IF (OP80_HMI_AutoMode AND NOT OP80_HMI_ManualMOde AND NOT OP80_HMI_StepMode) THEN
		OP80_Modeselection_FB.ModeWord:=1;
	ELSIF (NOT OP80_HMI_AutoMode AND OP80_HMI_ManualMOde AND NOT OP80_HMI_StepMode) THEN
		OP80_Modeselection_FB.ModeWord:=2;
	ELSIF  (NOT OP80_HMI_AutoMode AND NOT OP80_HMI_ManualMOde AND  OP80_HMI_StepMode) THEN
		OP80_Modeselection_FB.ModeWord:=3;
    ELSE   
		OP80_Modeselection_FB.ModeWord:=0;
END_IF
OP80_Modeselection_FB(
	ModeWord:= , 
	HomeConditionOK:=OP80_HomeConditionOK , 
	OperationEnable:=OP80_AutoSelected, 
	StartPB:=OP80_HMI_CycleStart , 
	SafetyAndNOError:= OP80_Safety_OK, 
	ModeAck:=TRUE , 
	HomingINProgress:=OP80_HomeRunning , 
	TempHomeOK:=OP80_Temp_hmeOK , 
	ResetPB:= , 
	AutoSelected=> OP80_AutoSelected, 
	ManualSelected=> OP80_ManualSelected, 
	StepSelected=>OP80_StepSelected , 
	ModeSelAck_Indication=> , 
	StatusDisplay=> , 
	AutoRunning:=OP80_AutoRunning, 
	StepRunning:=OP80_StepRunning , 
	StartEnable:=OP80_StartEnable  , 
	MachineStop:=OP80_Machine_Stop );

OP80_Safety_OK:=OperationEnable;	
	
IF OP80_AutoSelected OR OP80_ManualSelected AND NOT ( OP80_ErrorActive OR OP80_Safety_OK) THEN
	SR60_Vert_servo.bEnable:=TRUE;
ELSE
	SR60_Vert_servo.bEnable:=FALSE;
END_IF

IF SR80_Vert_servo.bAxisError OR NOT OP80_Safety_OK  THEN
	OP80_ErrorActive:=TRUE;
END_IF

OP80_Safety_OK:=OperationEnable;

IF OP80_Stop_Request AND NOT OP80_STN_ENABLE THEN
	OP80_Machine_Stop:=1;
END_IF
Gen_Timer(IN:=OP80_Machine_Stop,PT:=T#5S);
IF Gen_Timer.Q THEN
	OP80_Machine_Stop:=0;
END_IF

END_PROGRAM

// ---- POUs/Programs/OP80/OP80_MANUAL.TcPOU
PROGRAM OP80_MANUAL
VAR
	//SR80_Vert_servo_status:stManualModeAxis;
	SR80_Vert_servo_Axis :AXIS_REF;
    temp_safe:BOOL;
	enable:BOOL;
	reset:bool;
	Op80Enable: BOOL;
END_VAR


// IF MANUAL IS SELECTED 

//SR80_Vert_servo_ctrl.ABSmove_Start:=OP80_VERT_SERVO_STRT;
//OP80_SERVO_POS_DONE:= SR80_Vert_servo_ctrl.pos_done;

IF In_Range(SR80_Vert_servo_status.actualPosition,OP80_VERT_SERVO_SFE_WRK_POS,1) THEN
	OP80_SERVO_ON_SFE_WRK := TRUE;
ELSE
	OP80_SERVO_ON_SFE_WRK := FALSE;
END_IF

IF In_Range(SR80_Vert_servo_status.actualPosition,OP80_VERT_SERVO_HME_POS,1) THEN
	OP80_SERVO_ON_HOME := TRUE;
ELSE
	OP80_SERVO_ON_HOME := FALSE;
END_IF

IF In_Range(SR80_Vert_servo_status.actualPosition,OP80_VERT_SERVO_WRK_POS_1,1) THEN
	OP80_SERVO_ON_WRK_1 := TRUE;
ELSE
	OP80_SERVO_ON_WRK_1 := FALSE;
END_IF

IF In_Range(SR80_Vert_servo_status.actualPosition,OP80_VERT_SERVO_WRK_POS_2,1) THEN
	OP80_SERVO_ON_WRK_2 := TRUE;
ELSE
	OP80_SERVO_ON_WRK_2 := FALSE;
END_IF

OP80_VERT_SERVO_SFE_WRK_POS   :=  OP80_HMI_Safe_Work;
OP80_VERT_SERVO_HME_POS       :=  OP80_HMI_Safe_Home;
OP80_VERT_SERVO_WRK_POS_2     :=  OP80_VERT_SERVO_WORK_POS;
OP80_VERT_SERVO_WRK_POS_1	  := (OP80_VERT_SERVO_WRK_POS_2-OP80_HMI_Servo_Pos_Offset);

SR80_Vert_servo(
	bAxis1_Ref_Switch:= , 
	bInit:= , 
	bErrorReset:= OP80_HMI_Reset OR Servo_Reset , 
	bEnable:= Servo_Enable, 
	bMoveVelocity:= , 
	bHalt:= , 
	bManualMode:=OP80_ManualSelected AND MANUAL_SELECTED , 
	fHomePos:= , 
	fOverride:= , 
	fTargetPosition:=SR80_Vert_servo_ctrl.Position , 
	fTargetVelocity:=SR80_Vert_servo_ctrl.Velocity , 
	fAcc:= , 
	fDec:= , 
	Servo_High_Limit:= OP80_HMI_High_Limit,	
	Servo_Low_Limit:=  OP80_HMI_Low_Limit,	
	Safe_move_Conditions:=Servo_Safety,
	Axis:=SR80_Vert_servo_Axis  , 
	bmove_home:=SR80_Vert_servo_ctrl.Axis_Home_Cmd ,
	baxis_in_home_pos=>SR80_Vert_servo_ctrl.Axis_In_Home ,
	HME_WRITE_ADD:= 16#500F,	
	bHome:=SR80_Vert_servo_ctrl.Bsethome , 
	bSetPosition:=SR80_Vert_servo_ctrl.BsetPos , 
	bMoveAbsolute:=SR80_Vert_servo_ctrl.ABSmove_Start , 
	bMoveRelative:=SR80_Vert_servo_ctrl.RELmove_Start ,
	bMoveTorque :=SR80_Vert_servo_ctrl.Torque_mode_Start,
	stManualModeAxis:=SR80_Vert_servo_status , 
	sAxisState=>SR80_Vert_servo_ctrl.Axis_State , 
	bAxis_ready=>SR80_Vert_servo_ctrl.Axis_ready , 
	bAxisInPosition=> SR80_Vert_servo_ctrl.Axis_In_Pos, 
	bAxisError=>SR80_Vert_servo_ctrl.Axis_Error , 
	bAxisEnabled=> SR80_Vert_servo_ctrl.Axis_Enabled, 
	bAxisHomed=> SR80_Vert_servo_ctrl.Axis_reference, 
	bSetPositionDone=>   ,
    bsafe_to_move=>SR80_Vert_servo_ctrl.Safe_To_Move,  
	bABS_Pos_done=> SR80_Vert_servo_ctrl.pos_done,
	Actual_position=>SR80_Vert_servo_ctrl.Actual_Position ,  
	Actual_velocity=>SR80_Vert_servo_ctrl.Actual_Velocity , 
	Actual_Torque=> SR80_Vert_servo_ctrl.Actual_Torque,	
	bHaltDone=> , 
	bSTOPDone=> , 
	bHomeDone=> , 
	bDone=> );
	
IF MANUAL_SELECTED AND OP80_ManualSelected THEN
	SR80_Vert_servo_status.targetVelocity:=50;	
END_IF

OP80_LH_LVDT_VALUE := DINT_TO_REAL(OP80_LH)/10000;
OP80_RH_LVDT_VALUE := DINT_TO_REAL(OP80_RH)/10000;

END_PROGRAM

// ---- POUs/Programs/OP80/OP80_AUTOSEQUENCE.TcPOU
PROGRAM OP80_AUTOSEQUENCE
VAR

//INT

	OP80_FIXTURE_2					: INT;
	OP80_FIXTURE_1					: INT;	
	Dry_run : BOOL;
// TIMER
	OP80_AFT_WRK_POS : TON;
	
	check: BOOL;
	OP80_STN_MOVER: INT;
	OP80_Cycle_Time_FB : FB_Cycletime;
	MOVER_POS_RECHED_R: R_TRIG;
END_VAR

VAR PERSISTENT

END_VAR

IF (NOT OP80_AutoSelected) OR (OP80_ErrorActive OR OP80_HomeRunning ) OR NOT OperationEnable THEN
	OP80_AutoRunning:= FALSE;
	OP80_AutoSeq:= 10;
END_IF	


CASE OP80_AutoSeq OF
		
		10: IF (OP80_AutoSelected) THEN		// Check Automode Selected
				OP80_AutoSeq:=20;
	        END_IF
		
	    20:IF ( NOT OP80_ErrorActive) THEN		//Check No error
		       OP80_AutoSeq:=30;
      	   END_IF
		   
      	30:IF (NOT OP80_HomeRunning) THEN		//Check No Homerunning
      		   OP80_AutoSeq :=40;
      	   END_IF
		   
        40:IF (OP80_Main.OP80_Modeselection_FB.TempHomeOK)THEN	//Check Machine in Home
      		   OP80_AutoSeq:= 50;
      	   END_IF
		   
      	50:IF ( OP80_STN_ENABLE AND OP80_STN_RUNNING ) THEN		// Check Operation Completed Reset
      		   OP80_AutoSeq:=70;
		   ELSE
	   		   OP80_AutoSeq:=60;
      	   END_IF
		   
	   60:IF (AUTO_RUNNING OR (NOT AUTO_RUNNING AND OP80_HMI_CycleStart)) THEN		//Machine Start in Fully Automatic or Press Cycle Start For Semi Automatic
		    OP80_HomeConditionOK:=TRUE;
	 			IF( OP80_Main.OP80_Modeselection_FB.HomeConditionOK AND OP80_AutoSelected) THEN
					OP80_AutoRunning:=TRUE;
					OP80_StepRunning:= FALSE;		
				ELSIF (OP80_Main.OP80_Modeselection_FB.HomeConditionOK AND OP80_StepSelected) THEN
					OP80_AutoRunning:=FALSE;
					OP80_StepRunning:= TRUE;
				END_IF;
		  END_IF
		  
		  IF ((OP80_AutoRunning OR OP80_StepRunning) AND OP80_StartEnable) THEN
			OP80_AutoSeq:= 70;
		  END_IF	

      	70:  // SERVO POSITION SAFE CHECK
	       IF (OP80_SERVO_ON_SFE_WRK OR OP80_SERVO_ON_HOME) AND NOT SR80_Vert_servo_ctrl.ABSmove_Start THEN 
	        SR80_Vert_servo_ctrl.Position:=OP80_VERT_SERVO_WRK_POS_1;   
	        OP80_AutoSeq:=75;
	       END_IF
		   
		75: // WAITING FOR MOVER AND MOVING SERVO TO TARGET POSITION
			IF OP80_STN_ENABLE AND SR80_Vert_servo_ctrl.Position=OP80_VERT_SERVO_WRK_POS_1 THEN
			 SR80_Vert_servo_ctrl.Velocity:=OP80_HMI_Servo_Speed;
			 OP80_STN_RUNNING:=1;
			 SR80_Vert_servo_ctrl.ABSmove_Start:=TRUE;
			 IF OP80_FIXTURE_1=70 OR OP80_FIXTURE_2=70 THEN
			 	OP80_AutoSeq:=80;
			 ELSIF OP80_FIXTURE_1<>70 AND OP80_FIXTURE_2<>70 THEN
				OP80_AutoSeq:=76;
			 END_IF	
			END_IF

		 76:OP80_STN_ENABLE:=0;
			IF 	(MOVER_CMP_STATUS[OP80_STN_MOVER][1]=71 AND MOVER_CMP_STATUS[OP80_STN_MOVER][2]=71) THEN
				MOVER_STP_NO[OP80_CURR_MOVER]	:= (OP80_XTS_POS_NO*10);
			ELSE		
				STATION_DONE[OP80_CURR_MOVER][OP80_XTS_POS_NO]	:= TRUE;
			END_IF	
			IF MOVER_STP_NO[OP80_CURR_MOVER]<>((OP80_XTS_POS_NO*10)+1)THEN 
				OP80_CURR_MOVER	:= 0;
				OP80_AutoSeq	:= 76;  
			END_IF	
			
		80:  IF SR80_Vert_servo_ctrl.pos_done AND OP80_SERVO_ON_WRK_1 THEN
			   SR80_Vert_servo_ctrl.ABSmove_Start:=FALSE;
			   SR80_Vert_servo_ctrl.Position:=OP80_GVL.OP80_VERT_SERVO_WRK_POS_2;
			   SR80_Vert_servo_ctrl.Velocity:=(OP80_HMI_Servo_Speed-OP80_HMI_Servo_Speed_Offset);
			   OP80_AutoSeq:=90;
			 ELSIF SR80_Vert_servo_ctrl.pos_done AND OP80_SERVO_ON_WRK_2 THEN
 				OP80_AutoSeq:=100;
			 END_IF
			  
		90: IF OP80_SERVO_ON_WRK_1 AND NOT SR80_Vert_servo_ctrl.ABSmove_Start THEN                   
               SR80_Vert_servo_ctrl.ABSmove_Start:=TRUE;
				OP80_LH_LVDT_OK:=0;
				OP80_LH_LVDT_NOK:=0;
				OP80_RH_LVDT_OK:=0;
				OP80_RH_LVDT_NOK:=0; 
               OP80_AutoSeq:=100;
			END_IF
			
		100: // START THE SPINNER OK COMPONENT FIXTURE
			IF OP80_AFT_WRK_POS.Q AND OP80_SERVO_ON_WRK_2 THEN	
			 SR80_Vert_servo_ctrl.ABSmove_Start:=FALSE;		 
			  IF OP80_FIXTURE_1=70 THEN
			 	 IF In_Range(OP80_LH_LVDT_VALUE,OP80_SET_LVDT_VALUE,OP80_LVDT_TOLERANCE) THEN
				  OP80_LH_LVDT_OK  := 1;
				  OP80_LH_LVDT_NOK := 0;				  				  
			 	 ELSE
				  OP80_LH_LVDT_NOK := 1;
				  OP80_LH_LVDT_OK  := 0;
			 	 END_IF  
			  END_IF
			  IF OP80_FIXTURE_2=70 THEN
			  	IF In_Range(OP80_RH_LVDT_VALUE,OP80_SET_LVDT_VALUE,OP80_LVDT_TOLERANCE) THEN
				  OP80_RH_LVDT_OK  := 1;
				  OP80_RH_LVDT_NOK := 0;			  				  
			  	ELSE
				  OP80_RH_LVDT_NOK := 1;
				  OP80_RH_LVDT_OK  := 0;
			    END_IF
		 	  END_IF
				OP80_HMI_LH_LVDT_VALUE:=OP80_LH_LVDT_VALUE;
				OP80_HMI_RH_LVDT_VALUE:=OP80_RH_LVDT_VALUE;				  
			  IF NOT SR80_Vert_servo_ctrl.ABSmove_Start THEN
				 SR80_Vert_servo_ctrl.Position:=OP80_VERT_SERVO_SFE_WRK_POS;
				 SR80_Vert_servo_ctrl.Velocity:=OP80_HMI_Servo_Speed;
				 OP80_STN_ENABLE:=FALSE;
				 OP80_AutoSeq:=110;
			  END_IF				    			  
		    END_IF
			OP80_CURR_MOVER			:= OP80_STN_MOVER;
		
		110: // SERVO MOVE TO SAFE WORK POSITION	 
			IF NOT SR80_Vert_servo_ctrl.ABSmove_Start AND SR80_Vert_servo.fTargetPosition=OP80_VERT_SERVO_SFE_WRK_POS THEN
				SR80_Vert_servo_ctrl.ABSmove_Start:=TRUE;
				IF OP80_LH_LVDT_OK THEN
					MOVER_CMP_STATUS[OP80_CURR_MOVER][1]:=80;
				ELSIF OP80_LH_LVDT_NOK THEN  
					MOVER_CMP_STATUS[OP80_CURR_MOVER][1]:=81;	
				END_IF
				IF OP80_RH_LVDT_OK THEN
					MOVER_CMP_STATUS[OP80_CURR_MOVER][2]:=80;
				ELSIF OP80_RH_LVDT_NOK THEN  
					MOVER_CMP_STATUS[OP80_CURR_MOVER][2]:=81;	
				END_IF									
				OP80_AutoSeq:=120;
			END_IF

				
		120: // SERVO DONE
			IF SR80_Vert_servo_ctrl.pos_done AND OP80_SERVO_ON_SFE_WRK THEN
			 	SR80_Vert_servo_ctrl.ABSmove_Start:=FALSE;
				OP80_STN_ENABLE:=0;				
			 	OP80_AutoSeq:=70;
				OP80_STN_RUNNING:=0;
			IF (MOVER_CMP_STATUS[OP80_CURR_MOVER][1]=81 AND MOVER_CMP_STATUS[OP80_CURR_MOVER][2]=81) THEN	
				MOVER_STP_NO[OP80_CURR_MOVER]	:= (OP160_XTS_POS_NO*10);
			ELSE
			STATION_DONE[OP80_CURR_MOVER][OP80_XTS_POS_NO]			:= TRUE;
		   END_IF	
		END_IF		
END_CASE 

OP80_Cycle_Time_FB(i_b_startTime:=OP80_STN_ENABLE , i_b_stopTime:= NOT OP80_STN_ENABLE , o_t_StationTime=>OP80_Cycle_time );					


OP80_AFT_WRK_POS(IN:=(OP80_SERVO_ON_WRK_2 AND (OP80_AutoSeq=100)), PT:=INT_TO_TIME(OP80_DLY_AFT_SFE_WRK));

Dry_Run:=All_Station_Dry_Run;
IF Dry_run THEN
	OP80_FIXTURE_1:=70;
    OP80_FIXTURE_2:=70;
ELSE  
OP80_FIXTURE_1:=MOVER_CMP_STATUS[OP80_STN_MOVER][1];
OP80_FIXTURE_2:=MOVER_CMP_STATUS[OP80_STN_MOVER][2];	
END_IF


//############################		OP80 STATION ENABLE CONDITION		##########################

	OP80_STN_MOVER					:= MOVER_POSITION[OP80_XTS_POS_NO];
IF AUTO_WITH_XTS THEN
IF OP80_STN_MOVER>0 THEN
IF NOT(END_OF_CYCLE AND MOVER_CMP_STATUS[OP80_STN_MOVER][1]=5 AND MOVER_CMP_STATUS[OP80_STN_MOVER][2]=5)THEN	
	OP80_STN_ENABLE					:= MOVER_POS_RECHED[OP80_STN_MOVER] AND ((MOVER_CMP_STATUS[OP80_STN_MOVER][1]=70)OR 
										(MOVER_CMP_STATUS[OP80_STN_MOVER][2]=70)) AND STATION_ENABLE_CONTROL;
ELSE
	STATION_DONE[OP80_STN_MOVER][OP80_XTS_POS_NO]			:= TRUE;	
END_IF
ELSE
	OP80_STN_ENABLE										:= FALSE;
END_IF		
END_IF

END_PROGRAM

// ---- POUs/Programs/OP80/OP80_ERROR.TcPOU
PROGRAM OP80_ERROR
VAR
	OP80_StepErr_1: TON;
	OP80_Step_Err_2: TON;
END_VAR

// Set ERROR ACTIVE
IF ((OP80_GVL.OP80_ErrorWord_0<>0) OR (OP80_GVL.OP80_ErrorWord_1<>0) OR (OP80_GVL.OP80_ErrorWord_2<>0)) THEN
	OP80_GVL.OP80_ErrorActive:= TRUE;
	END_IF

//Reset ErrorActive
IF (OP80_HMI_Reset OR HMI_Reset) THEN 
	OP80_GVL.OP80_ErrorActive:= FALSE;
	OP80_GVL.OP80_ErrorWord_0:= 0;
	OP80_GVL.OP80_ErrorWord_1:= 0;
	OP80_GVL.OP80_ErrorWord_2:= 0;

END_IF

OP80_ErrorWord_0.0:=SR80_Vert_servo.bAxisError;
OP80_ErrorWord_0.1:=NOT OperationEnable;

// Auto Seq Step Error
//Servo not reaching work position
OP80_StepErr_1(IN:=(OP80_AutoSeq=80) , PT:=T#5S , Q=> , ET=> );
IF (OP80_AutoSeq=80 AND NOT OP80_GVL.OP80_SERVO_ON_WRK_1 AND OP80_StepErr_1.Q) THEN
	OP80_GVL.OP80_ErrorWord_0.2:=TRUE;
END_IF

// Servo Not Reached home position or safe-work position
OP80_Step_Err_2(IN:=OP80_AutoSeq=120 , PT:=T#5S , Q=> , ET=> );
IF (OP80_AutoSeq=120 AND NOT SR80_Vert_servo_ctrl.Axis_In_Home AND OP80_Step_Err_2.Q) THEN
	OP80_GVL.OP80_ErrorWord_0.3:=TRUE;
END_IF

//OP20_StepErr_3(IN:=( OP80_HomeRunning AND (OP80_Homing_Seq=10)), PT:=T#5S , Q=> , ET=> );
//IF OP20_StepErr_3.Q THEN
//	OP20_GVL.OP20_ErrorWord_0.4:=TRUE;
//END_IF

END_PROGRAM

// ---- POUs/Programs/OP80/OP80_Initialization_Seq.TcPOU
PROGRAM OP80_Initialization_Seq
VAR
END_VAR

IF (SR80_Vert_servo_ctrl.Axis_In_Home)THEN
    OP80_Temp_hmeOK:=TRUE;
	OP80_HomeRunning:=FALSE;
	OP80_Homing_Seq:=0;
ELSE
	OP80_Temp_hmeOK:=FALSE;	
END_IF

CASE OP80_Homing_Seq OF
	0: IF (OP80_AutoSelected AND NOT OP80_HomeRunning AND NOT OP80_ErrorActive AND NOT  OP80_AutoRunning AND NOT OP80_StepRunning AND NOT OP80_Temp_hmeOK ) THEN
		OP80_HomeRunning:=TRUE;
		OP80_Homing_Seq:=10;	
	   END_IF
	   
	10:IF (OP80_HomeRunning AND (OP80_HMI_Homing OR HMI_Reset))THEN 
		IF (SR80_Vert_servo_ctrl.Axis_In_Home) THEN 
			OP80_Homing_Seq:=20;
			SR80_Vert_servo_ctrl.Axis_Home_Cmd:=FALSE;
		ELSE
			SR80_Vert_servo_ctrl.Position:=0;
			SR80_Vert_servo_ctrl.Velocity:=100;
			SR80_Vert_servo_ctrl.ABSmove_Start:=TRUE;
			SR80_Vert_servo_ctrl.Axis_Home_Cmd:=TRUE;
	    END_IF
	   END_IF
	
	20:	OP80_Homing_Seq:=0;
		OP80_HomeRunning:=FALSE;
	
END_CASE

END_PROGRAM

// ---- POUs/Programs/OP80/op80_toolchangeover.TcPOU
PROGRAM op80_toolchangeover
VAR
	op80_tool_change                    : tool_changeover;
	OP80_TOOL_CHANGE_MODE_SELECTED      : BOOL;
	fb_reset_1                          : BOOL;
	tool_6_fb                           : BOOL;
	tool_8_fb                           : BOOL;
	OP80_TOL_UNLOD_STRT					: BOOL;
	OP80_TOL_LOAD_STRT					: BOOL;
	OP80_TOL_DISENGAGE					: BOOL;
	OP80_TOL_ENGAGE						: BOOL;
	op80_manual_lock                    : BOOL;
	op80_manual_unlock                  : BOOL;
	OP80_UNLD_STUS                      : STRING;
	OP80_LOAD_STUS                      : STRING;
	op80_t2_manual_lock: BOOL;
END_VAR

VAR PERSISTENT
	
	OP80_TOL_WRK_POS					: LREAL;
	OP80_TOL_HME_POS					: LREAL;
	op80_TOL_VELOCITY					: LREAL;
	OP80_TOL_CHNGE_CMPLE				: BOOL;
	OP80_TOL_LOAD_COMPLE                : BOOL;
	OP80_TOL_UNLOAD_COMPLE              : BOOL;
	
END_VAR

IF OP80_TOOL_CHANGE_MODE_SELECTED THEN

op80_tool_change(
	actual_pos:= SR80_Vert_servo_ctrl.Actual_Position , 
	actual_vel:= SR80_Vert_servo_ctrl.Actual_Velocity, 
	target_work_pos:= OP80_TOL_WRK_POS, 
	target_home_pos:= OP80_TOL_HME_POS, 
	target_vel_from_hmi:= op80_TOL_VELOCITY, 
	station_number:= , 
	mover_number:= , 
	no_of_mover_present:= , 
	model_selected:= model_selected, 
	tool_unloading_start:=OP80_TOL_UNLOD_STRT , 
	tool_loading_start:=OP80_TOL_LOAD_STRT , 
	error_active:= , 
	station_in_auto:= OP80_AutoSelected,                   
	station_in_home:=  ,                                   
	absoulte_move_done:= SR80_Vert_servo_ctrl.Axis_In_Pos, 
	tool_6_3_present:= tool_6_fb, 
	tool_7_89_present:= tool_8_fb, 
	fb_reset:=fb_reset_1,
	SERVO_TOL_CHECK_OFFSET_POS := 18, 
	tool_changer_over_complete=> OP80_TOL_CHNGE_CMPLE,
	tool_disengage=> OP80_TOL_DISENGAGE, 
	tool_engagae=> OP80_TOL_ENGAGE, 
	tool_loading_complete=> OP80_TOL_LOAD_COMPLE, 
	tool_unloading_complete=> OP80_TOL_UNLOAD_COMPLE, 
	servo_move_abs=>SR80_Vert_servo_ctrl.ABSmove_Start, 
	unloading_status=>OP80_UNLD_STUS , 
	loading_status=>OP80_LOAD_STUS , 
	target_pos_to_servo=> SR80_Vert_servo_ctrl.Position, 
	target_vel_to_servo=> SR80_Vert_servo_ctrl.Velocity,
    tool_loading_failed := );
	
END_IF	

IF op80_manual_lock OR OP80_TOL_ENGAGE THEN
	O80_TOOL_CHO_UNLOCK_Q1153_0 :=0;
	O80_TOOL_CHO_LOCK_Q1153_1   :=1;
ELSIF op80_manual_unlock OR OP80_TOL_DISENGAGE THEN
	  O80_TOOL_CHO_LOCK_Q1153_1    :=0;
	  O80_TOOL_CHO_UNLOCK_Q1153_0  :=1;
END_IF

END_PROGRAM

// ---- POUs/Programs/OP90/OP90_MAIN.TcPOU
PROGRAM OP90_MAIN
VAR


END_VAR


OP90_MANUAL();
OP90_SERVO();
OP90_AUTO();
OP90_CAMERA();
OP90_Camera_FB();
//OP90_LH_CONVEYOR();
//OP90_RH_CONVEYOR();
OP90_HOMING();
OP90_Conveyor_FBs();

IF OP90_SRV_RH_VERT.bAxisError OR OP90_SRV_LH_VERT.bAxisError OR OP90_GUIDE_SERVO.bAxisError OR OP90_SRV_HORZ.bAxisError OR OP90A_CYLINDER_ERR<>0 THEN
	OP90_ERR			:= TRUE;
ELSE
	OP90_ERR			:= FALSE;
END_IF
///////////////////////////////////////////////////////////////////////////////////
// WILL BE DELETED
//	1)OP90_DRY_RUN

OP90_MODE_BLOCK(
	ModeWord:= OP90_MODE_WORD, 
	HomeConditionOK:= OP90_ALL_HOME, 
	OperationEnable:= OperationEnable, 
	StartPB:= OP90_STRT_PB, 
	SafetyAndNOError:= NOT OP90_ERR, 
	ModeAck:= 1, 
	HomingINProgress:= , 
	TempHomeOK:= , 
	ResetPB:= OP90_RESET_PB, 
	AutoSelected=> OP90_AUTO_SELECTED, 
	ManualSelected=> OP90_MANUAL_SELECTED, 
	StepSelected=> OP90_STEP_SELECTED, 
	ModeSelAck_Indication=> , 
	StatusDisplay=> , 
	AutoRunning:=OP90_AUTO_RUNNING, 
	StepRunning:=OP90_STEP_RUNNING , 
	StartEnable:=OP90_START_ENABLE , 
	MachineStop:=OP90_MACHINE_STOP );

END_PROGRAM

// ---- POUs/Programs/OP90/OP90_MANUAL.TcPOU
PROGRAM OP90_MANUAL
VAR
// VISION
	OP90_M_VISIN1_LGT						: BOOL;
	OP90_H_VISIN1_LGT						: BOOL;
	OP90_M_VISIN2_LGT						: BOOL;
	OP90_H_VISIN2_LGT						: BOOL;
// DOOR
	OP90_M_LH_DOOR							: BOOL;
	OP90_H_LH_DOOR							: BOOL;
	OP90_M_RH_DOOR							: BOOL;
	OP90_H_RH_DOOR							: BOOL;
	OP90_M_FRNT_DOOR						: BOOL;
	OP90_H_FRNT_DOOR						: BOOL;
	OP90_M_BCK_DOOR							: BOOL;
	OP90_H_BCK_DOOR							: BOOL;



	
// CYLINDER FB MAPPING
							(*INT*)
	OP90_LH_GRP_STATS						: INT;
	OP90_RH_GRP_STATS						: INT;
	OP90_POS1_LCK_CYL_STUS					: INT;
	OP90_POS2_LCK_CYL_STUS					: INT;
	OP90_POS_SLIDE_CYL_STUS					: INT;
	OP90_SUP_HORZP1_CYL_STUS				: INT;
	OP90_SUP_VERTP1_CYL_STUTS				: INT;
	OP90_SUP_HORZP2_CYL_STUS				: INT;
	OP90_SUP_VERTP2_CYL_STUS				: INT;
	OP90_LH_REJP1_CYL_STUS					: INT;
	OP90_RH_REJP1_CYL_STUS					: INT;
	OP90_LH_REJP2_CYL_STUS					: INT;
	OP90_RH_REJP2_CYL_STUS					: INT;
							(*ALARM*)
	OP90_LH_GRIPPER_A1						: BOOL;
	OP90_LH_GRIPPER_A2						: BOOL;
	OP90_LH_GRIPPER_A3						: BOOL;
	OP90_LH_GRIPPER_A4						: BOOL;
	OP90_LH_GRIPPER_A5						: BOOL;
	OP90_RH_GRIPPER_A1						: BOOL;
	OP90_RH_GRIPPER_A2						: BOOL;
	OP90_RH_GRIPPER_A3						: BOOL;
	OP90_RH_GRIPPER_A4						: BOOL;
	OP90_RH_GRIPPER_A5						: BOOL;
	OP90_POS1_LCK_CYL_A1					: BOOL;
	OP90_POS1_LCK_CYL_A2					: BOOL;
	OP90_POS1_LCK_CYL_A3					: BOOL;
	OP90_POS1_LCK_CYL_A4					: BOOL;
	OP90_POS1_LCK_CYL_A5					: BOOL;
	OP90_POS2_LCK_CYL_A1					: BOOL;
	OP90_POS2_LCK_CYL_A2					: BOOL;
	OP90_POS2_LCK_CYL_A3					: BOOL;
	OP90_POS2_LCK_CYL_A4					: BOOL;
	OP90_POS2_LCK_CYL_A5					: BOOL;
	OP90_POS_SLIDE_CYL_A1					: BOOL;
	OP90_POS_SLIDE_CYL_A2					: BOOL;
	OP90_POS_SLIDE_CYL_A3					: BOOL;
	OP90_POS_SLIDE_CYL_A4					: BOOL;
	OP90_POS_SLIDE_CYL_A5					: BOOL;
	OP90_SUP_HORZP1_CYL_A1					: BOOL;
	OP90_SUP_HORZP1_CYL_A2					: BOOL;
	OP90_SUP_HORZP1_CYL_A3					: BOOL;
	OP90_SUP_HORZP1_CYL_A4					: BOOL;
	OP90_SUP_HORZP1_CYL_A5					: BOOL;
	OP90_SUP_VERTP1_CYL_A1					: BOOL;
	OP90_SUP_VERTP1_CYL_A2					: BOOL;
	OP90_SUP_VERTP1_CYL_A3					: BOOL;
	OP90_SUP_VERTP1_CYL_A4					: BOOL;
	OP90_SUP_VERTP1_CYL_A5					: BOOL;
	OP90_SUP_HORZP2_CYL_A1					: BOOL;
	OP90_SUP_HORZP2_CYL_A2					: BOOL;
	OP90_SUP_HORZP2_CYL_A3					: BOOL;
	OP90_SUP_HORZP2_CYL_A4					: BOOL;
	OP90_SUP_HORZP2_CYL_A5					: BOOL;
	OP90_SUP_VERTP2_CYL_A1					: BOOL;
	OP90_SUP_VERTP2_CYL_A2					: BOOL;
	OP90_SUP_VERTP2_CYL_A3					: BOOL;
	OP90_SUP_VERTP2_CYL_A4					: BOOL;
	OP90_SUP_VERTP2_CYL_A5					: BOOL;
	OP90_LH_REJP1_CYL_A1					: BOOL;
	OP90_LH_REJP1_CYL_A2					: BOOL;
	OP90_LH_REJP1_CYL_A3					: BOOL;
	OP90_LH_REJP1_CYL_A4					: BOOL;
	OP90_LH_REJP1_CYL_A5					: BOOL;
	OP90_RH_REJP1_CYL_A1					: BOOL;
	OP90_RH_REJP1_CYL_A2					: BOOL;
	OP90_RH_REJP1_CYL_A3					: BOOL;
	OP90_RH_REJP1_CYL_A4					: BOOL;
	OP90_RH_REJP1_CYL_A5					: BOOL;
	OP90_LH_REJP2_CYL_A1					: BOOL;
	OP90_LH_REJP2_CYL_A2					: BOOL;
	OP90_LH_REJP2_CYL_A3					: BOOL;
	OP90_LH_REJP2_CYL_A4					: BOOL;
	OP90_LH_REJP2_CYL_A5					: BOOL;
	OP90_RH_REJP2_CYL_A1					: BOOL;
	OP90_RH_REJP2_CYL_A2					: BOOL;
	OP90_RH_REJP2_CYL_A3					: BOOL;
	OP90_RH_REJP2_CYL_A4					: BOOL;
	OP90_RH_REJP2_CYL_A5					: BOOL;
							(*BOOL*)

	OP90_M_LH_GRP_MANUALPB1					: BOOL;
	OP90_M_LH_GRP_MANUALPB2					: BOOL;
	OP90_M_RH_GRP_MANUALPB1					: BOOL;
	OP90_M_RH_GRP_MANUALPB2					: BOOL;
	OP90_M_POS1_LCK_HOME					: BOOL;
	OP90_M_POS1_LCK_WORK					: BOOL;
	OP90_M_POS2_LCK_HOME					: BOOL;
	OP90_M_POS2_LCK_WORK					: BOOL;
	OP90_M_MVE_POS1							: BOOL;
	OP90_M_MVE_POS2							: BOOL;
	OP90_M_MVR_SUP_HORZP1_HOME				: BOOL;
	OP90_M_MVR_SUP_HORZP1_WRK				: BOOL;
	OP90_M_MVR_SUP_VERTP1_HOME				: BOOL;
	OP90_M_MVR_SUP_VERTP1_WRK				: BOOL;
	OP90_M_LH_REJP1_HOME					: BOOL;
	OP90_M_LH_REJP1_WRK						: BOOL;
	OP90_M_RH_REJP1_HOME					: BOOL;
	OP90_M_RH_REJP1_WRK						: BOOL;
	OP90_M_MVR_SUP_HORZP2_HOME				: BOOL;
	OP90_M_MVR_SUP_HORZP2_WRK				: BOOL;
	OP90_M_MVR_SUP_VERTP2_HOME				: BOOL;
	OP90_M_MVR_SUP_VERTP2_WRK				: BOOL;
	OP90_M_LH_REJP2_HOME					: BOOL;
	OP90_M_LH_REJP2_WRK						: BOOL;
	OP90_M_RH_REJP2_HOME					: BOOL;
	OP90_M_RH_REJP2_WRK						: BOOL;
	OP90_M_LH_AIR_PURGE						: BOOL;
	OP90_H_LH_AIR_PURGE						: BOOL;
	OP90_M_RH_AIR_PURGE						: BOOL;
	OP90_H_RH_AIR_PURGE						: BOOL;

	TEMPPR: BOOL;








	Temp3: BOOL;
	Temp4: BOOL;
	OP90_MOVER_HOME: BOOL;
END_VAR

IF OP90_MANUAL_SELECTED THEN
	
OP90_M_VISIN1_LGT								:=	OP90_H_VISIN1_LGT; 		 // Q400.0 VISION 1 MANUAL ON
OP90_M_VISIN2_LGT								:=	OP90_H_VISIN2_LGT; 	 	 // Q400.1 VISION 2 MANUAL ON
OP90_M_LH_DOOR 									:= 	OP90_H_LH_DOOR;			// Q400.2 LH DOOR MANUAL ON
OP90_M_RH_DOOR 									:= 	OP90_H_RH_DOOR;			// Q400.3 RH DOOR MANUAL ON
OP90_M_FRNT_DOOR 								:= 	OP90_H_FRNT_DOOR;		// Q400.4 FRONT DOOR MANUAL ON
OP90_M_BCK_DOOR 								:= 	OP90_H_BCK_DOOR;		// Q400.5 BACK DOOR MANUAL ON
OP90_M_LH_AIR_PURGE								:=  OP90_H_LH_AIR_PURGE;		// Q1250.4 REJECTION AIR PURGE
OP90_M_RH_AIR_PURGE								:=  OP90_H_RH_AIR_PURGE;		// Q1251.2 REJECTION AIR PURGE


CASE OP90_CYL_NUM OF
	
	1: IF OP90_HOME THEN
		OP90_M_LH_GRP_MANUALPB1					:=TRUE;
		OP90_M_LH_GRP_MANUALPB2					:=FALSE;
		END_IF                      			
		IF OP90_WORK THEN           			
		OP90_M_LH_GRP_MANUALPB2					:=TRUE;
		OP90_M_LH_GRP_MANUALPB1					:=FALSE;
		END_IF                              	
		                                    	
	2:  IF OP90_HOME THEN                   	
		OP90_M_RH_GRP_MANUALPB1					:=TRUE;
		OP90_M_RH_GRP_MANUALPB2					:=FALSE;
		END_IF                      			
		IF OP90_WORK THEN           			
		OP90_M_RH_GRP_MANUALPB2					:=TRUE;
		OP90_M_RH_GRP_MANUALPB1					:=FALSE;
		END_IF                      		
		                            		
	3: IF OP90_HOME THEN            		
		OP90_M_POS1_LCK_HOME					:=TRUE;
		OP90_M_POS1_LCK_WORK					:=FALSE;
		END_IF                      			
		IF OP90_WORK THEN           			
		OP90_M_POS1_LCK_WORK					:=TRUE;
		OP90_M_POS1_LCK_HOME					:=FALSE;
		END_IF                      			
		                            			
	4: IF OP90_HOME THEN            			
		OP90_M_POS2_LCK_HOME					:=TRUE;
		OP90_M_POS2_LCK_WORK					:=FALSE;
		END_IF                      			
		IF OP90_WORK THEN           			
		OP90_M_POS2_LCK_WORK					:=TRUE;
		OP90_M_POS2_LCK_HOME					:=FALSE;
		END_IF                              	
		                                    	
	5: IF OP90_HOME THEN                    	
		OP90_M_MVE_POS1							:=TRUE;
		OP90_M_MVE_POS2							:=FALSE;
		END_IF                      		
		IF OP90_WORK THEN           		
		OP90_M_MVE_POS2							:=TRUE;
		OP90_M_MVE_POS1							:=FALSE;
		END_IF                              	
		                                    	
	6: 	IF OP90_HOME THEN                   	
		OP90_M_MVR_SUP_HORZP1_HOME				:=TRUE;
		OP90_M_MVR_SUP_HORZP1_WRK				:=FALSE;
		END_IF                      			
		IF OP90_WORK THEN           			
		OP90_M_MVR_SUP_HORZP1_WRK				:=TRUE;
		OP90_M_MVR_SUP_HORZP1_HOME				:=FALSE;
		END_IF                      			
	                                			
	7: 	IF OP90_HOME THEN           			
		OP90_M_MVR_SUP_VERTP1_HOME				:=TRUE;
		OP90_M_MVR_SUP_VERTP1_WRK				:=FALSE;
		END_IF                      			
		IF OP90_WORK THEN           	    	
		OP90_M_MVR_SUP_VERTP1_WRK				:=TRUE;
		OP90_M_MVR_SUP_VERTP1_HOME				:=FALSE;
		END_IF                              	
		                                    	
	8: 	IF OP90_HOME THEN                   	
		OP90_M_LH_REJP1_HOME					:=TRUE;
		OP90_M_LH_REJP1_WRK						:=FALSE;
		END_IF                      		
		IF OP90_WORK THEN           		
		OP90_M_LH_REJP1_WRK						:=TRUE;
		OP90_M_LH_REJP1_HOME					:=FALSE;
		END_IF                      			
		                            			
	9: IF OP90_HOME THEN            			
		OP90_M_RH_REJP1_HOME					:=TRUE;
		OP90_M_RH_REJP1_WRK						:=FALSE;
		END_IF                      			
		IF OP90_WORK THEN           			
		OP90_M_RH_REJP1_WRK						:=TRUE;
		OP90_M_RH_REJP1_HOME					:=FALSE;
		END_IF                      			
		                            			
	10: IF OP90_HOME THEN           			
		OP90_M_MVR_SUP_HORZP2_HOME				:=TRUE;
		OP90_M_MVR_SUP_HORZP2_WRK				:=FALSE;
		END_IF                      			
		IF OP90_WORK THEN           			
		OP90_M_MVR_SUP_HORZP2_WRK				:=TRUE;
		OP90_M_MVR_SUP_HORZP2_HOME				:=FALSE;
		END_IF
		
	11:	IF OP90_HOME THEN
		OP90_M_MVR_SUP_VERTP2_HOME				:=TRUE;
		OP90_M_MVR_SUP_VERTP2_WRK				:=FALSE;
		END_IF                      			
		IF OP90_WORK THEN           			
		OP90_M_MVR_SUP_VERTP2_WRK				:=TRUE;
		OP90_M_MVR_SUP_VERTP2_HOME				:=FALSE;
		END_IF                      			
		                            			
	12: IF OP90_HOME THEN           			
		OP90_M_LH_REJP2_HOME					:=TRUE;
		OP90_M_LH_REJP2_WRK						:=FALSE;
		END_IF                      			
		IF OP90_WORK THEN           			
		OP90_M_LH_REJP2_WRK						:=TRUE;
		OP90_M_LH_REJP2_HOME					:=FALSE;
		END_IF                      			
		                            			
	13: IF OP90_HOME THEN           			
		OP90_M_RH_REJP2_HOME					:=TRUE;
		OP90_M_RH_REJP2_WRK						:=FALSE;
		END_IF                      			
		IF OP90_WORK THEN           			
		OP90_M_RH_REJP2_WRK						:=TRUE;
		OP90_M_RH_REJP2_HOME					:=FALSE;
		END_IF 	
	
END_CASE

CASE OP90_SERVO_NUM OF
	
	1: 	OP90_SRV_HORZ_STATUS.jogPos				:=OP90_JOG_POS AND NOT OP90_JOG_NEG;
		OP90_SRV_HORZ_STATUS.jogNeg				:=OP90_JOG_NEG AND NOT OP90_JOG_POS;
		OP90_SRV_HORZ_CNTRL.Axis_Home_Cmd		:=OP90_SET_HME;
		OP90_SRV_HORZ_STATUS.targetPositon		:=OP90_TRGT_POS;
//       OP90_SRV_HORZ_STATUS.targetVelocity 	:=OP90_TRGT_VEL; 
		OP90_SRV_HORZ_STATUS.moveAbsolute		:=OP90_MOVE_TARGT;
		OP90_SERVO_ACTUAL_POS					:=DINT_TO_LREAL(LREAL_TO_DINT(OP90_SRV_HORZ_STATUS.actualPosition*100))/100;
        OP90_SERVO_FAULT						:=OP90_SRV_HORZ.bAxisError;
		OP90_HOME_REFERENCE						:=OP90_SRV_HORZ_CNTRL.Axis_reference;
		OP90_M_SERVO_ENABLE						:=OP90_SRV_HORZ.bAxisEnabled;

         
	2:  OP90_SRV_LH_VERT_STATUS.jogPos			:=OP90_JOG_POS AND NOT OP90_JOG_NEG;
		OP90_SRV_LH_VERT_STATUS.jogNeg			:=OP90_JOG_NEG AND NOT OP90_JOG_POS;
		OP90_SRV_LH_VERT_CNTRL.Axis_Home_Cmd	:=OP90_SET_HME;
		OP90_SRV_LH_VERT_STATUS.targetPositon	:=OP90_TRGT_POS;
//		OP90_SRV_LH_VERT_STATUS.targetVelocity	:=OP90_TRGT_VEL; 
		OP90_SRV_LH_VERT_STATUS.moveAbsolute	:=OP90_MOVE_TARGT;
		OP90_SERVO_ACTUAL_POS					:=DINT_TO_LREAL(LREAL_TO_DINT(OP90_SRV_LH_VERT_STATUS.actualPosition*100))/100;
        OP90_SERVO_FAULT						:=OP90_SRV_LH_VERT.bAxisError;
		OP90_HOME_REFERENCE						:=OP90_SRV_LH_VERT_CNTRL.Axis_reference;		
		OP90_M_SERVO_ENABLE						:=OP90_SRV_LH_VERT.bAxisEnabled;
	
		
	3:  OP90_SRV_RH_VERT_STATUS.jogPos			:=OP90_JOG_POS AND NOT OP90_JOG_NEG;
		OP90_SRV_RH_VERT_STATUS.jogNeg			:=OP90_JOG_NEG AND NOT OP90_JOG_POS;
		OP90_SRV_RH_VERT_CNTRL.Axis_Home_Cmd	:=OP90_SET_HME;
		OP90_SRV_RH_VERT_STATUS.targetPositon	:=OP90_TRGT_POS;
//		OP90_SRV_RH_VERT_STATUS.targetVelocity	:=OP90_TRGT_VEL; 
		OP90_SRV_RH_VERT_STATUS.moveAbsolute	:=OP90_MOVE_TARGT;
		OP90_SERVO_ACTUAL_POS					:=DINT_TO_LREAL(LREAL_TO_DINT(OP90_SRV_RH_VERT_STATUS.actualPosition*100))/100;
        OP90_SERVO_FAULT						:=OP90_SRV_RH_VERT.bAxisError;
		OP90_HOME_REFERENCE						:=OP90_SRV_RH_VERT_CNTRL.Axis_reference;
		OP90_M_SERVO_ENABLE						:=OP90_SRV_RH_VERT.bAxisEnabled;
	
	4: OP90_STP_LH_ROTRY_STATUS.jogPos			:=OP90_JOG_POS AND NOT OP90_JOG_NEG;
	   OP90_STP_LH_ROTRY_STATUS.jogNeg      	:=OP90_JOG_NEG AND NOT OP90_JOG_POS;
		OP90_STP_LH_ROTRY_CNTRL.Axis_Home_Cmd	:=OP90_SET_HME;
		OP90_STP_LH_ROTRY_STATUS.targetPositon	:=OP90_TRGT_POS;
//		OP90_STP_LH_ROTRY_STATUS.targetVelocity	:=OP90_TRGT_VEL;
		OP90_STP_LH_ROTRY_STATUS.moveAbsolute	:=OP90_MOVE_TARGT;
		OP90_SERVO_ACTUAL_POS					:=DINT_TO_LREAL(LREAL_TO_DINT(OP90_STP_LH_ROTRY_STATUS.actualPosition*100))/100;
        OP90_SERVO_FAULT						:=OP90_LH_SRV_ROTRY.bAxisError;
		OP90_HOME_REFERENCE						:=OP90_STP_LH_ROTRY_CNTRL.Axis_reference;		
		OP90_M_SERVO_ENABLE						:=1;		

	   
	5: OP90_STP_RH_ROTRY_STATUS.jogPos			:=OP90_JOG_POS AND NOT OP90_JOG_NEG;
	   OP90_STP_RH_ROTRY_STATUS.jogNeg      	:=OP90_JOG_NEG AND NOT OP90_JOG_POS;
	   OP90_STP_RH_ROTRY_CNTRL.Axis_Home_Cmd	:=OP90_SET_HME;
		OP90_STP_RH_ROTRY_STATUS.targetPositon	:=OP90_TRGT_POS;	   
//		OP90_STP_RH_ROTRY_STATUS.targetVelocity	:=OP90_TRGT_VEL;	   
		OP90_STP_RH_ROTRY_STATUS.moveAbsolute	:=OP90_MOVE_TARGT;
		OP90_SERVO_ACTUAL_POS					:=DINT_TO_LREAL(LREAL_TO_DINT(OP90_STP_RH_ROTRY_STATUS.actualPosition*100))/100;
        OP90_SERVO_FAULT						:=OP90_RH_SRV_ROTRY.bAxisError;
		OP90_HOME_REFERENCE						:=OP90_STP_RH_ROTRY_CNTRL.Axis_reference;
		OP90_M_SERVO_ENABLE						:=1;
	   
	   
		
	6: OP90_GIUDE_SER_STATUS.jogPos				:=OP90_JOG_POS AND NOT OP90_JOG_NEG;
	   OP90_GIUDE_SER_STATUS.jogNeg         	:=OP90_JOG_NEG AND NOT OP90_JOG_POS;
	   OP90_SERVO_GUIDE_CNTRL.Axis_Home_Cmd		:=OP90_SET_HME;
		OP90_GIUDE_SER_STATUS.targetPositon		:=OP90_TRGT_POS;	 	   
//		OP90_GIUDE_SER_STATUS.targetVelocity	:=OP90_TRGT_VEL;	 	   
		OP90_GIUDE_SER_STATUS.moveAbsolute		:=OP90_MOVE_TARGT;	 	   
		OP90_SERVO_ACTUAL_POS					:=DINT_TO_LREAL(LREAL_TO_DINT(OP90_GIUDE_SER_STATUS.actualPosition*100))/100;
        OP90_SERVO_FAULT						:=OP90_GUIDE_SERVO.bAxisError;
		OP90_HOME_REFERENCE						:=OP90_SERVO_GUIDE_CNTRL.Axis_reference;
 		OP90_M_SERVO_ENABLE						:=OP90_GUIDE_SERVO.bAxisEnabled;
		
	   
	7: OP90_SRV_LH_CNVY_STATUS.jogPos			:=OP90_JOG_POS AND NOT OP90_JOG_NEG;
	   OP90_SRV_LH_CNVY_STATUS.jogNeg       	:=OP90_JOG_NEG AND NOT OP90_JOG_POS;
	   OP90_SRV_LH_CNVY_CNTRL.Axis_Home_Cmd		:=OP90_SET_HME;
		OP90_SRV_LH_CNVY_STATUS.targetPositon	:=OP90_TRGT_POS;		   
//		OP90_SRV_LH_CNVY_STATUS.targetVelocity	:=OP90_TRGT_VEL;	   
		OP90_SRV_LH_CNVY_STATUS.moveAbsolute	:=OP90_MOVE_TARGT;
		OP90_SERVO_ACTUAL_POS					:=DINT_TO_LREAL(LREAL_TO_DINT(OP90_SRV_LH_CNVY_STATUS.actualPosition*100))/100;
        OP90_SERVO_FAULT						:=OP90_LH_CNVY.bAxisError;
		OP90_HOME_REFERENCE						:=OP90_SRV_LH_CNVY_CNTRL.Axis_reference;
		OP90_M_SERVO_ENABLE						:=1;
		
	   
	   
		
	8: OP90_SRV_RH_CNVY_STATUS.jogPos			:=OP90_JOG_POS AND NOT OP90_JOG_NEG;	 
	   OP90_SRV_LH_CNVY_STATUS.jogNeg       	:=OP90_JOG_NEG AND NOT OP90_JOG_POS;
	   OP90_SRV_RH_CNVY_CNTRL.Axis_Home_Cmd		:=OP90_SET_HME;
		OP90_SRV_RH_CNVY_STATUS.targetPositon	:=OP90_TRGT_POS;	
//		OP90_SRV_RH_CNVY_STATUS.targetVelocity	:=OP90_TRGT_VEL;	
		OP90_SRV_RH_CNVY_STATUS.moveAbsolute	:=OP90_MOVE_TARGT;
		OP90_SERVO_ACTUAL_POS					:=DINT_TO_LREAL(LREAL_TO_DINT(OP90_SRV_RH_CNVY_STATUS.actualPosition*100))/100;
        OP90_SERVO_FAULT						:=OP90_RH_CNVY.bAxisError;
		OP90_HOME_REFERENCE						:=OP90_SRV_LH_CNVY_CNTRL.Axis_reference;	
		OP90_M_SERVO_ENABLE						:=1;	                           
 
END_CASE


ELSE
// VISION, DOOR, AIRPURGE
OP90_M_VISIN1_LGT								:= FALSE;
OP90_M_VISIN2_LGT								:= FALSE;
OP90_M_LH_DOOR 									:= FALSE;
OP90_M_RH_DOOR 	                				:= FALSE;
OP90_M_FRNT_DOOR  		        				:= FALSE;
OP90_M_BCK_DOOR                 				:= FALSE;
OP90_M_LH_AIR_PURGE								:= FALSE;
OP90_M_RH_AIR_PURGE								:= FALSE;

// CYLINDER
OP90_M_LH_GRP_MANUALPB1							:= FALSE;
OP90_M_LH_GRP_MANUALPB2							:= FALSE;
OP90_M_RH_GRP_MANUALPB2							:= FALSE;
OP90_M_RH_GRP_MANUALPB1							:= FALSE;
OP90_M_POS1_LCK_WORK							:= FALSE;
OP90_M_POS1_LCK_HOME							:= FALSE;
OP90_M_POS2_LCK_WORK							:= FALSE;
OP90_M_POS2_LCK_HOME            				:= FALSE;
OP90_M_MVE_POS2									:= FALSE;
OP90_M_MVE_POS1									:= FALSE;
OP90_M_MVR_SUP_HORZP1_WRK	 					:= FALSE;
OP90_M_MVR_SUP_HORZP1_HOME 						:= FALSE;
OP90_M_MVR_SUP_VERTP1_WRK	  					:= FALSE;
OP90_M_MVR_SUP_VERTP1_HOME  					:= FALSE;
OP90_M_LH_REJP1_HOME							:= FALSE;
OP90_M_LH_REJP1_WRK								:= FALSE;
OP90_M_RH_REJP1_WRK								:= FALSE;
OP90_M_RH_REJP1_HOME  							:= FALSE;
OP90_M_MVR_SUP_HORZP2_HOME						:= FALSE;
OP90_M_MVR_SUP_HORZP2_WRK 						:= FALSE;
OP90_M_MVR_SUP_VERTP2_HOME						:= FALSE;
OP90_M_MVR_SUP_VERTP2_WRK						:= FALSE;
OP90_M_LH_REJP2_HOME							:= FALSE;
OP90_M_LH_REJP2_WRK								:= FALSE;
OP90_M_RH_REJP2_WRK								:= FALSE;
OP90_M_RH_REJP2_HOME  							:= FALSE;

END_IF

// CYLINDER FUNTIONAL BLOCK

OP90_LH_GRIPPER(													// OP90_LH_GRIPPER_CYLINDER_FB
	Auto:= OP90_AUTO_RUNNING OR OP90_STEP_RUNNING, 
	Manual:= OP90_MANUAL_SELECTED, 
	ErrorActive:= OP90_ERR, 
	ResetPB:= OP90_RESET_PB, 									
	Sensor1:= I90_RET_LH_GRIPR_CYL_CLSE_I1200_0,                                             
	Sensor2:= I90_RET_LH_GRIPR_CYL_OPN_I1200_1 OR OP90_LH_GRP_BYPASS,
	ManualPB1:= OP90_M_LH_GRP_MANUALPB1, 
	ManualPB2:= OP90_M_LH_GRP_MANUALPB2, 
	AutoCmd1:= OP90_A_LH_GRP_AUTCMD1, 
	AutoCmd2:= OP90_A_LH_GRP_AUTCMD2, 
	OperationEnable:= OperationEnable, 
	SafeHome:=1, 
	SafeWork:=1, 
	HomingCmd1:= OP90_LH_GRP_HOMING1, 
	Pulse_1Sec:= Pulse_Block.Q1Hz, 
	BlinkingBit:= , 
	TimeOut1:= 5, 
	TimeOut2:= 5, 
	TimeOut3:= 5, 
	Solenoid1=> O90_RET_LH_GRIPR_CYL_CLSE_Q1240_0, 
	Solenoid2=> O90_RET_LH_GRIPR_CYL_OPN_Q1240_1, 
	AlarmSensor1=> OP90_LH_GRIPPER_A1, 
	AlarmSensor2=> OP90_LH_GRIPPER_A2, 
	AlarmSolenoid1=> OP90_LH_GRIPPER_A3, 
	AlarmSolenoid2=> OP90_LH_GRIPPER_A4, 
	AllSignal=> OP90_LH_GRIPPER_A5, 
	AlarmPresent=> OP90A_CYLINDER_ERR.0, 
	Position1=> , 
	Position2=> , 
	HomeSensorBlink=> , 
	WorkSensorBlink=> , 
	Status:=OP90_LH_GRP_STATS );
	
	
OP90_RH_GRIPPER(													//OP90_RH_GRIPPER_CYLINDER_FB
	Auto:= OP90_AUTO_RUNNING OR OP90_STEP_RUNNING, 
	Manual:= OP90_MANUAL_SELECTED, 
	ErrorActive:= OP90_ERR, 
	ResetPB:= OP90_RESET_PB, 
	Sensor1:= I90_RET_RH_GRIPR_CYL_CLSE_I1200_2, 
	Sensor2:= I90_RET_RH_GRIPR_CYL_OPN_I1200_3 OR OP90_RH_GRP_BYPASS, 
	ManualPB1:= OP90_M_RH_GRP_MANUALPB1, 
	ManualPB2:= OP90_M_RH_GRP_MANUALPB2, 
	AutoCmd1:= OP90_A_RH_GRP_AUTCMD1, 
	AutoCmd2:= OP90_A_RH_GRP_AUTCMD2, 
	OperationEnable:= OperationEnable, 
	SafeHome:= 1, 
	SafeWork:= 1, 
	HomingCmd1:= OP90_RH_GRP_HOMING1, 
	Pulse_1Sec:= Pulse_Block.Q1Hz, 
	BlinkingBit:= , 
	TimeOut1:= 5, 
	TimeOut2:= 5, 
	TimeOut3:= 5,
	Solenoid1=> O90_RET_RH_GRIPR_CYL_CLSE_Q1240_2, 
	Solenoid2=> O90_RET_RH_GRIPR_CYL_OPN_Q1240_3, 
	AlarmSensor1=> OP90_RH_GRIPPER_A1, 
	AlarmSensor2=> OP90_RH_GRIPPER_A2, 
	AlarmSolenoid1=> OP90_RH_GRIPPER_A3, 
	AlarmSolenoid2=> OP90_RH_GRIPPER_A4, 
	AllSignal=> OP90_RH_GRIPPER_A5, 
	AlarmPresent=> OP90A_CYLINDER_ERR.1, 
	Position1=> , 
	Position2=> , 
	HomeSensorBlink=> , 
	WorkSensorBlink=> , 
	Status:=OP90_RH_GRP_STATS );

//OP90_POS1_LCK_CYLINDER_SAFE_WRK/HOME
	
	OP90_POS1_LCK_CYL.SafeWork	:= OP90_POS_SLIDE_CYL.Sensor2 OR OP90_POS_SLIDE_CYL.Sensor1;

OP90_POS1_LCK_CYL(														//OP90_POS1_LCK_CYLINDER_FB
	Auto:= OP90_AUTO_RUNNING OR OP90_STEP_RUNNING, 
	Manual:= OP90_MANUAL_SELECTED, 
	ErrorActive:= OP90_ERR, 
	ResetPB:= OP90_RESET_PB, 
	Sensor1:= NOT O90_POS_LOCK_CYL2_VLVE_2_Q1240_7, 												//O90_POS_LOCK_CYL1_VLVE_1_Q1240_4
	Sensor2:= O90_POS_LOCK_CYL2_VLVE_2_Q1240_7, 
	ManualPB1:= OP90_M_POS1_LCK_HOME, 
	ManualPB2:= OP90_M_POS1_LCK_WORK, 
	AutoCmd1:= , 
	AutoCmd2:= , 
	OperationEnable:= OperationEnable AND Temp3, 
	SafeHome:= TRUE, 
	SafeWork:= , 
	HomingCmd1:= , 
	Pulse_1Sec:= Pulse_Block.Q1Hz, 
	BlinkingBit:= , 
	TimeOut1:= 5, 
	TimeOut2:= 5, 
	TimeOut3:= 5,
	Solenoid1=> , 												//O90_POS_LOCK_CYL1_VLVE_1_Q1240_4
	Solenoid2=> O90_POS_LOCK_CYL2_VLVE_2_Q1240_7, 
	AlarmSensor1=> OP90_POS1_LCK_CYL_A1, 
	AlarmSensor2=> OP90_POS1_LCK_CYL_A2, 
	AlarmSolenoid1=> OP90_POS1_LCK_CYL_A3, 
	AlarmSolenoid2=> OP90_POS1_LCK_CYL_A4, 
	AllSignal=> OP90_POS1_LCK_CYL_A5, 
	AlarmPresent=>OP90A_CYLINDER_ERR.2 , 
	Position1=> , 
	Position2=> , 
	HomeSensorBlink=> , 
	WorkSensorBlink=> , 
	Status:=OP90_POS1_LCK_CYL_STUS );

//OP90_POS2_LCK_CYLINDER_SAFE_WRK/HOME
	
	OP90_POS2_LCK_CYL.SafeWork	:= OP90_POS_SLIDE_CYL.Sensor2 OR OP90_POS_SLIDE_CYL.Sensor1;	
	
OP90_POS2_LCK_CYL(														//OP90_OP90_POS2_LCK_CYLINDER_FB
	Auto:= OP90_AUTO_RUNNING OR OP90_STEP_RUNNING, 
	Manual:= OP90_MANUAL_SELECTED, 
	ErrorActive:= OP90_ERR, 
	ResetPB:= OP90_RESET_PB, 
	Sensor1:= NOT O90_POS_LOCK_CYL1_VLVE_2_Q1240_5, 													//O90_POS_LOCK_CYL2_VLVE_1_Q1240_6
	Sensor2:= O90_POS_LOCK_CYL1_VLVE_2_Q1240_5, 
	ManualPB1:= OP90_M_POS2_LCK_HOME, 
	ManualPB2:= OP90_M_POS2_LCK_WORK, 
	AutoCmd1:= , 
	AutoCmd2:= , 
	OperationEnable:= OperationEnable AND Temp3, 
	SafeHome:= TRUE, 
	SafeWork:=, 
	HomingCmd1:= , 
	Pulse_1Sec:= Pulse_Block.Q1Hz, 
	BlinkingBit:= , 
	TimeOut1:= 5, 
	TimeOut2:= 5, 
	TimeOut3:= 5,
	Solenoid1=> , 												//O90_POS_LOCK_CYL2_VLVE_1_Q1240_6
	Solenoid2=> O90_POS_LOCK_CYL1_VLVE_2_Q1240_5,
	AlarmSensor1=> OP90_POS2_LCK_CYL_A1, 
	AlarmSensor2=> OP90_POS2_LCK_CYL_A2, 
	AlarmSolenoid1=> OP90_POS2_LCK_CYL_A3, 
	AlarmSolenoid2=> OP90_POS2_LCK_CYL_A4, 
	AllSignal=> OP90_POS2_LCK_CYL_A5, 
	AlarmPresent=>OP90A_CYLINDER_ERR.3 , 
	Position1=> , 
	Position2=> , 
	HomeSensorBlink=> , 
	WorkSensorBlink=> , 
	Status:= OP90_POS2_LCK_CYL_STUS);
	
//OP90_POS_SLIDE_CYLINDER_SAFE_WRK/HOME
	OP90_POS_SLIDE_CYL.SafeHome	:= OP90_POS2_LCK_CYL.Sensor1 AND OP90_POS1_LCK_CYL.Sensor1;
	OP90_POS_SLIDE_CYL.SafeWork := OP90_POS2_LCK_CYL.Sensor1 AND OP90_POS1_LCK_CYL.Sensor1;
	
OP90_POS_SLIDE_CYL(													//OP90_POS_SLIDE_CYLINDER_FB
	Auto:= OP90_AUTO_SELECTED OR OP90_STEP_SELECTED, 
	Manual:= OP90_MANUAL_SELECTED, 
	ErrorActive:= OP90_ERR, 
	ResetPB:= OP90_RESET_PB, 
	Sensor1:= I90_POSTN_SLIDE_CYL_FWD_I1200_5, 
	Sensor2:= I90_POSTN_SLIDE_CYL_REV_I1200_4, 
	ManualPB1:= OP90_M_MVE_POS1, 
	ManualPB2:= OP90_M_MVE_POS2, 
	AutoCmd1:= OP90_POS_SLIDE_CYL.auto AND OP90_POS1_V6_3, 
	AutoCmd2:= OP90_POS_SLIDE_CYL.auto AND OP90_POS2_V7_89, 
	OperationEnable:= OperationEnable, 
	SafeHome:=1, 
	SafeWork:=1, 
	HomingCmd1:= , 
	Pulse_1Sec:= Pulse_Block.Q1Hz, 
	BlinkingBit:= , 
	TimeOut1:= 5, 
	TimeOut2:= 5, 
	TimeOut3:= 5, 
	Solenoid1=> O90_POSTN_SLIDE_CYL_REV_Q1241_0, 
	Solenoid2=> O90_POSTN_SLIDE_CYL_FWD_Q1241_1, 
	AlarmSensor1=> OP90_POS_SLIDE_CYL_A1, 
	AlarmSensor2=> OP90_POS_SLIDE_CYL_A2, 
	AlarmSolenoid1=> OP90_POS_SLIDE_CYL_A3, 
	AlarmSolenoid2=> OP90_POS_SLIDE_CYL_A4, 
	AllSignal=> OP90_POS_SLIDE_CYL_A5, 
	AlarmPresent=> OP90A_CYLINDER_ERR.4, 
	Position1=> , 
	Position2=> , 
	HomeSensorBlink=> , 
	WorkSensorBlink=> , 
	Status:= OP90_POS_SLIDE_CYL_STUS);

//OP90_SUP_HORZP1_CYLINDER_SAFE_WRK/HOME
	OP90_SUP_HORZP1_CYL.SafeHome := OP90_SUP_VERTP1_CYL.Sensor1;
	OP90_SUP_HORZP1_CYL.SafeWork := OP90_SUP_VERTP1_CYL.Sensor1;(* AND OP90_MOVER_HOME ;*)
	
OP90_SUP_HORZP1_CYL(													//OP90_SUP_HORZP1_CYLINDER_FB
	Auto:= OP90_AUTO_RUNNING OR OP90_STEP_RUNNING, 
	Manual:= OP90_MANUAL_SELECTED, 
	ErrorActive:= OP90_ERR, 
	ResetPB:= OP90_RESET_PB, 
	Sensor1:= I90_LH_MOVR_SUP_HORZ_CYL_REV_I1201_0, 
	Sensor2:= I90_LH_MOVR_SUP_HORZ_CYL_FWD_I1201_1, 
	ManualPB1:= OP90_M_MVR_SUP_HORZP1_HOME, 	
	ManualPB2:= OP90_M_MVR_SUP_HORZP1_WRK, 	
	AutoCmd1:= OP90_A_MVR_SUP_HORZP1_HME, 
	AutoCmd2:= OP90_A_MVR_SUP_HORZP1_WRK, 
	OperationEnable:= OperationEnable, 
	SafeHome:= , 
	SafeWork:= , 
	HomingCmd1:= OP90_SUP_HORZP1_CYL_HOME1, 
	Pulse_1Sec:= Pulse_Block.Q1Hz, 
	BlinkingBit:= , 
	TimeOut1:= 5, 
	TimeOut2:= 5, 
	TimeOut3:= 5,
	Solenoid1=>  O90_RH_MOVR_SUP_HORZ_CYL_REV_Q1242_0,  
	Solenoid2=>  O90_RH_MOVR_SUP_HORZ_CYL_FWD_Q1242_1 , 
	AlarmSensor1=> OP90_SUP_HORZP1_CYL_A1, 
	AlarmSensor2=> OP90_SUP_HORZP1_CYL_A2, 
	AlarmSolenoid1=> OP90_SUP_HORZP1_CYL_A3, 
	AlarmSolenoid2=> OP90_SUP_HORZP1_CYL_A4, 
	AllSignal=> OP90_SUP_HORZP1_CYL_A5, 
	AlarmPresent=> OP90A_CYLINDER_ERR.5, 
	Position1=> , 
	Position2=> , 
	HomeSensorBlink=> , 
	WorkSensorBlink=> , 
	Status:= OP90_SUP_HORZP1_CYL_STUS);

//OP90_SUP_VERTP1_CYLINDER_SAFE_WRK/HME

	OP90_SUP_VERTP1_CYL.SafeHome := OP90_SUP_HORZP1_CYL.Sensor1 OR OP90_SUP_HORZP1_CYL.Sensor2;
	OP90_SUP_VERTP1_CYL.SafeWork := OP90_SUP_HORZP1_CYL.Sensor1 OR OP90_SUP_HORZP1_CYL.Sensor2;

OP90_SUP_VERTP1_CYL(												//OP90_SUP_VERTP1_CYLINDER_FB
	Auto:= OP90_AUTO_RUNNING OR OP90_STEP_RUNNING, 
	Manual:= OP90_MANUAL_SELECTED, 
	ErrorActive:= OP90_ERR, 
	ResetPB:= OP90_RESET_PB, 
	Sensor1:=  I90_RH_MOVR_SUP_VERT_CYL_DWN_I1201_2, 
	Sensor2:=  I90_RH_MOVR_SUP_VERT_CYL_UP_I1201_3, 
	ManualPB1:= OP90_M_MVR_SUP_VERTP1_HOME,	 
	ManualPB2:= OP90_M_MVR_SUP_VERTP1_WRK,	 
	AutoCmd1:= OP90_A_MVR_SUP_VERTP1_HME, 
	AutoCmd2:= OP90_A_MVR_SUP_VERTP1_WRK, 
	OperationEnable:= OperationEnable, 
	SafeHome:= , 
	SafeWork:= , 
	HomingCmd1:= OP90_SUP_VERTP1_CYL_HOME1, 
	Pulse_1Sec:= Pulse_Block.Q1Hz, 
	BlinkingBit:= , 
	TimeOut1:= 5, 
	TimeOut2:= 5, 
	TimeOut3:= 5, 
	Solenoid1=> O90_RH_MOVR_SUP_VERT_CYL_DWN_Q1241_6, 
	Solenoid2=> O90_RH_MOVR_SUP_VERT_CYL_UP_Q1241_7 , 
	AlarmSensor1=> OP90_SUP_VERTP1_CYL_A1, 
	AlarmSensor2=> OP90_SUP_VERTP1_CYL_A2, 
	AlarmSolenoid1=> OP90_SUP_VERTP1_CYL_A3, 
	AlarmSolenoid2=> OP90_SUP_VERTP1_CYL_A4, 
	AllSignal=> OP90_SUP_VERTP1_CYL_A5, 
	AlarmPresent=> OP90A_CYLINDER_ERR.6, 
	Position1=> , 
	Position2=> , 
	HomeSensorBlink=> , 
	WorkSensorBlink=> , 
	Status:= OP90_SUP_VERTP1_CYL_STUTS);

//OP90_SUP_HORZP2_CYLINDER_SAFE_WRK/HOME
	OP90_SUP_HORZP2_CYL.SafeHome := OP90_SUP_VERTP2_CYL.Sensor1;
	OP90_SUP_HORZP2_CYL.SafeWork := OP90_SUP_VERTP2_CYL.Sensor1;(* AND OP90_MOVER_HOME ;*)
	
OP90_SUP_HORZP2_CYL(															//OP90_SUP_HORZP2_CYLINDER_FB
	Auto:= OP90_AUTO_RUNNING OR OP90_STEP_RUNNING, 
	Manual:= OP90_MANUAL_SELECTED, 
	ErrorActive:= OP90_ERR, 
	ResetPB:= OP90_RESET_PB, 
	Sensor1:= I90_RH_MOVR_SUP_HORZ_CYL_REV_I1201_4, 
	Sensor2:= I90_RH_MOVR_SUP_HORZ_CYL_FWD_I1201_5, 
	ManualPB1:= OP90_M_MVR_SUP_HORZP2_HOME,
	ManualPB2:= OP90_M_MVR_SUP_HORZP2_WRK, 
	AutoCmd1:= OP90_A_MVR_SUP_HORZP2_HME,  
	AutoCmd2:= OP90_A_MVR_SUP_HORZP2_WRK,  
	OperationEnable:= OperationEnable, 
	SafeHome:= , 
	SafeWork:= , 
	HomingCmd1:= OP90_SUP_HORZP2_CYL_HOME1, 
	Pulse_1Sec:= Pulse_Block.Q1Hz, 
	BlinkingBit:= , 
	TimeOut1:= 5, 
	TimeOut2:= 5, 
	TimeOut3:= 5,
	Solenoid1=>O90_LH_MOVR_SUP_HORZ_CYL_REV_Q1241_4,
	Solenoid2=>O90_LH_MOVR_SUP_HORZ_CYL_FWD_Q1241_5, 
	AlarmSensor1=> OP90_SUP_HORZP2_CYL_A1, 
	AlarmSensor2=> OP90_SUP_HORZP2_CYL_A2, 
	AlarmSolenoid1=> OP90_SUP_HORZP2_CYL_A3, 
	AlarmSolenoid2=> OP90_SUP_HORZP2_CYL_A4, 
	AllSignal=> OP90_SUP_HORZP2_CYL_A5, 
	AlarmPresent=>OP90A_CYLINDER_ERR.7 , 
	Position1=> , 
	Position2=> , 
	HomeSensorBlink=> , 
	WorkSensorBlink=> , 
	Status:= OP90_SUP_HORZP2_CYL_STUS);

//OP90_SUP_VERTP1_CYLINDER_SAFE_WRK/HME

	OP90_SUP_VERTP2_CYL.SafeHome := OP90_SUP_HORZP2_CYL.Sensor1 OR OP90_SUP_HORZP2_CYL.Sensor2;
	OP90_SUP_VERTP2_CYL.SafeWork := OP90_SUP_HORZP2_CYL.Sensor1 OR OP90_SUP_HORZP2_CYL.Sensor2;
	
OP90_SUP_VERTP2_CYL(
	Auto:= OP90_AUTO_RUNNING OR OP90_STEP_RUNNING, 
	Manual:= OP90_MANUAL_SELECTED, 
	ErrorActive:= OP90_ERR, 
	ResetPB:= OP90_RESET_PB, 
	Sensor1:= I90_LH_MOVR_SUP_VERT_CYL_DWN_I1200_6,
	Sensor2:= I90_LH_MOVR_SUP_VERT_CYL_UP_I1200_7, 
	ManualPB1:= OP90_M_MVR_SUP_VERTP2_HOME,
	ManualPB2:= OP90_M_MVR_SUP_VERTP2_WRK, 
	AutoCmd1:= OP90_A_MVR_SUP_VERTP2_HME, 
	AutoCmd2:= OP90_A_MVR_SUP_VERTP2_WRK, 
	OperationEnable:= OperationEnable, 
	SafeHome:= , 
	SafeWork:= , 
	HomingCmd1:= OP90_SUP_VERTP2_CYL_HOME1, 
	Pulse_1Sec:= Pulse_Block.Q1Hz, 
	BlinkingBit:= , 
	TimeOut1:= 5, 
	TimeOut2:= 5, 
	TimeOut3:= 5, 
	Solenoid1=>  O90_LH_MOVR_SUP_VERT_CYL_DWN_Q1241_2,
	Solenoid2=>   O90_LH_MOVR_SUP_VERT_CYL_UP_Q1241_3,
	AlarmSensor1=> OP90_SUP_VERTP2_CYL_A1, 
	AlarmSensor2=> OP90_SUP_VERTP2_CYL_A2, 
	AlarmSolenoid1=> OP90_SUP_VERTP2_CYL_A3, 
	AlarmSolenoid2=> OP90_SUP_VERTP2_CYL_A4, 
	AllSignal=> OP90_SUP_VERTP2_CYL_A5, 
	AlarmPresent=> OP90A_CYLINDER_ERR.8, 
	Position1=> , 
	Position2=> , 
	HomeSensorBlink=> , 
	WorkSensorBlink=> , 
	Status:= OP90_SUP_VERTP2_CYL_STUS);
	
OP90_LH_REJP1_CYL(														//OP90_LH_REJP1_CYLINDER_FB
	Auto:= OP90_AUTO_SELECTED OR OP90_STEP_RUNNING, 
	Manual:= OP90_MANUAL_SELECTED, 
	ErrorActive:= OP90_ERR, 
	ResetPB:= OP90_RESET_PB, 
	Sensor1:= I90_LH1_REJ_SLIDE_FWD_I1210_1, 
	Sensor2:= I90_LH1_REJ_SLIDE_REV_I1210_0 , 
	ManualPB1:= OP90_M_LH_REJP1_HOME, 
	ManualPB2:= OP90_M_LH_REJP1_WRK, 	
	AutoCmd1:= OP90_A_LH_REJP1_HOME, 
	AutoCmd2:= OP90_A_LH_REJP1_WORK, 
	OperationEnable:= OperationEnable, 
	SafeHome:= 1, 
	SafeWork:= 1, 
	HomingCmd1:= , 
	Pulse_1Sec:= Pulse_Block.Q1Hz, 
	BlinkingBit:= , 
	TimeOut1:= 5, 
	TimeOut2:= 5, 
	TimeOut3:= 5, 
	Solenoid1=> O90_LH1_REJ_SLIDE_FWD_Q1250_1, 
	Solenoid2=> O90_LH1_REJ_SLIDE_REV_Q1250_0, 
	AlarmSensor1=> OP90_LH_REJP1_CYL_A1, 
	AlarmSensor2=> OP90_LH_REJP1_CYL_A2, 
	AlarmSolenoid1=> OP90_LH_REJP1_CYL_A3, 
	AlarmSolenoid2=> OP90_LH_REJP1_CYL_A4, 
	AllSignal=> OP90_LH_REJP1_CYL_A5, 
	AlarmPresent=> OP90A_CYLINDER_ERR.9, 
	Position1=> , 
	Position2=> , 
	HomeSensorBlink=> , 
	WorkSensorBlink=> , 
	Status:= OP90_LH_REJP1_CYL_STUS);
	
OP90_RH_REJP1_CYL(													//OP90_RH_REJP1_CYLINDER_FB
	Auto:= OP90_AUTO_SELECTED OR OP90_STEP_RUNNING, 
	Manual:= OP90_MANUAL_SELECTED, 
	ErrorActive:= OP90_ERR, 
	ResetPB:= OP90_RESET_PB, 
	Sensor1:= I90_RH1_REJ_SLIDE_FWD_I1210_3, 
	Sensor2:= I90_RH1_REJ_SLIDE_REV_I1210_2, 
	ManualPB1:= OP90_M_RH_REJP1_HOME, 
	ManualPB2:= OP90_M_RH_REJP1_WRK,  
	AutoCmd1:= OP90_A_RH_REJP1_HOME, 
	AutoCmd2:= OP90_A_RH_REJP1_WORK, 
	OperationEnable:= OperationEnable, 
	SafeHome:= 1, 
	SafeWork:= 1, 
	HomingCmd1:= , 
	Pulse_1Sec:= Pulse_Block.Q1Hz, 
	BlinkingBit:= , 
	TimeOut1:= 5, 
	TimeOut2:= 5, 
	TimeOut3:= 5, 
	Solenoid1=> O90_RH1_REJ_SLIDE_FWD_Q1250_3, 
	Solenoid2=> O90_RH1_REJ_SLIDE_REV_Q1250_2, 
	AlarmSensor1=> OP90_RH_REJP1_CYL_A1, 
	AlarmSensor2=> OP90_RH_REJP1_CYL_A2, 
	AlarmSolenoid1=> OP90_RH_REJP1_CYL_A3, 
	AlarmSolenoid2=> OP90_RH_REJP1_CYL_A4, 
	AllSignal=> OP90_RH_REJP1_CYL_A5, 
	AlarmPresent=> OP90A_CYLINDER_ERR.10, 
	Position1=> , 
	Position2=> , 
	HomeSensorBlink=> , 
	WorkSensorBlink=> , 
	Status:= OP90_RH_REJP1_CYL_STUS);
	
OP90_LH_REJP2_CYL(														//OP90_LH_REJP2_CYLINDER_FB
	Auto:= OP90_AUTO_SELECTED OR OP90_STEP_RUNNING, 
	Manual:= OP90_MANUAL_SELECTED, 
	ErrorActive:= OP90_ERR, 
	ResetPB:= OP90_RESET_PB, 
	Sensor1:= I90_LH2_REJ_SLIDE_REV_I1210_4 , 
	Sensor2:= I90_LH2_REJ_SLIDE_FWD_I1210_5 , 
	ManualPB1:= OP90_M_LH_REJP2_HOME, 
	ManualPB2:= OP90_M_LH_REJP2_WRK,  
	AutoCmd1:= OP90_A_LH_REJP2_HOME, 
	AutoCmd2:= OP90_A_LH_REJP2_WORK, 
	OperationEnable:= OperationEnable, 
	SafeHome:=1 , 
	SafeWork:= 1, 
	HomingCmd1:= , 
	Pulse_1Sec:= Pulse_Block.Q1Hz, 
	BlinkingBit:= , 
	TimeOut1:= 5, 
	TimeOut2:= 5, 
	TimeOut3:= 5, 
	Solenoid1=> O90_LH2_REJ_SLIDE_REV_Q1250_6, 
	Solenoid2=>  O90_LH2_REJ_SLIDE_FWD_Q1250_7, 
	AlarmSensor1=> OP90_LH_REJP2_CYL_A1, 
	AlarmSensor2=> OP90_LH_REJP2_CYL_A2, 
	AlarmSolenoid1=> OP90_LH_REJP2_CYL_A3, 
	AlarmSolenoid2=> OP90_LH_REJP2_CYL_A4, 
	AllSignal=> OP90_LH_REJP2_CYL_A5, 
	AlarmPresent=>OP90A_CYLINDER_ERR.11 , 
	Position1=> , 
	Position2=> , 
	HomeSensorBlink=> , 
	WorkSensorBlink=> , 
	Status:= OP90_LH_REJP2_CYL_STUS);
	
OP90_RH_REJP2_CYL(															//OP90_RH_REJP2_CYLINDER_FB
	Auto:= OP90_AUTO_SELECTED OR OP90_STEP_RUNNING, 
	Manual:= OP90_MANUAL_SELECTED, 
	ErrorActive:= OP90_ERR, 
	ResetPB:= OP90_RESET_PB, 
	Sensor1:= I90_RH2_REJ_SLIDE_REV_I1210_6, 
	Sensor2:= I90_RH2_REJ_SLIDE_FWD_I1210_7, 
	ManualPB1:= OP90_M_RH_REJP2_HOME, 
	ManualPB2:= OP90_M_RH_REJP2_WRK,  
	AutoCmd1:= OP90_A_RH_REJP2_HOME, 
	AutoCmd2:= OP90_A_RH_REJP2_WORK, 
	OperationEnable:= OperationEnable, 
	SafeHome:= 1, 
	SafeWork:= 1, 
	HomingCmd1:= , 
	Pulse_1Sec:= Pulse_Block.Q1Hz, 
	BlinkingBit:= , 
	TimeOut1:= 5, 
	TimeOut2:= 5, 
	TimeOut3:= 5, 
	Solenoid1=> O90_RH2_REJ_SLIDE_REV_Q1251_0, 
	Solenoid2=> O90_RH2_REJ_SLIDE_FWD_Q1251_1, 
	AlarmSensor1=> OP90_RH_REJP2_CYL_A1, 
	AlarmSensor2=> OP90_RH_REJP2_CYL_A2, 
	AlarmSolenoid1=> OP90_RH_REJP2_CYL_A3, 
	AlarmSolenoid2=> OP90_RH_REJP2_CYL_A4, 
	AllSignal=> OP90_RH_REJP2_CYL_A5, 
	AlarmPresent=> OP90A_CYLINDER_ERR.12, 
	Position1=> , 
	Position2=> , 
	HomeSensorBlink=> , 
	WorkSensorBlink=> , 
	Status:= OP90_RH_REJP2_CYL_STUS);

END_PROGRAM

// ---- POUs/Programs/OP90/OP90_SERVO.TcPOU
PROGRAM OP90_SERVO
VAR
// STRING
	OP90_SRV_LH_VERT_FB					: STRING;
	OP90_SRV_RH_VERT_FB					: STRING;
	OP90_SRV_GUID_STOPER_FB				: STRING;	
	OP90_SRV_HORZ_FB					: STRING;	
// BOOL
	OP90_MOVER_SAFE						: BOOL;
	OP90_BLCK_INITZ						: BOOL;
	NOT_REF								: BOOL;
	FESTO_NOT_NEED						: BOOL;
	Conv_Contrl: BOOL;
	Conv_Contrl1: BOOL;
	OP90_LH_ROTARY_STUTS: STRING;
	OP90_RH_ROTARY_STUTS: STRING;
END_VAR

VAR PERSISTENT
	

	OP90_HORZ_WRK_SPD					: LREAL;
	OP90_HORZ_HME_SPD					: LREAL;
END_VAR

//////////////////////////////////////OP90_HORZ WRK_HOME///////////////////////////////////
IF OP90_A_SRV_HORZ_WRK AND NOT OP90_A_SRV_HORZ_HME AND OP90_SRV_LH_VRT_HME_FB AND OP90_SRV_RH_VRT_HME_FB THEN
	OP90_SRV_HORZ_CNTRL.ABSmove_Start		:= TRUE;
	OP90_SRV_HORZ_CNTRL.Position			:= OP90_SRV_HORZ_WRK_MM ;
	OP90_SRV_LIMIT.OP90_A_HORZ_VELOCITY		:= OP90_HORZ_WRK_SPD;
IF OP90_SRV_HORZ_WRK_FB THEN
	OP90_A_SRV_HORZ_WRK						:= FALSE;
	OP90_SRV_HORZ_CNTRL.ABSmove_Start		:= FALSE;
END_IF
END_IF

IF OP90_A_SRV_HORZ_HME AND NOT OP90_A_SRV_HORZ_WRK AND OP90_SRV_LH_VRT_HME_FB AND OP90_SRV_RH_VRT_HME_FB THEN
	OP90_SRV_HORZ_CNTRL.ABSmove_Start		:= TRUE;
	OP90_SRV_HORZ_CNTRL.Position			:= OP90_SRV_HORZ_HME_MM ;
	OP90_SRV_LIMIT.OP90_A_HORZ_VELOCITY		:= OP90_HORZ_HME_SPD;
IF OP90_SRV_HORZ_HME_FB THEN
	OP90_A_SRV_HORZ_HME						:= FALSE;
	OP90_SRV_HORZ_CNTRL.ABSmove_Start		:= FALSE;
END_IF
END_IF
/////////////////////////////////////////OP90_LH VRT HMR WRK///////////////////////////////
IF OP90_A_SRV_LHVERT_HME AND NOT OP90_A_SRV_LHVERT_PCKWRK AND NOT OP90_A_SRV_LHVERT_SPLCWRK AND NOT OP90_A_SRV_LHVERT_PLCWRK THEN
	OP90_SRV_LH_VERT_CNTRL.ABSmove_Start	:= TRUE;
	OP90_SRV_LH_VERT_CNTRL.Position			:= OP90_SRV_VERT_LH_HME_MM ;
IF OP90_SRV_LH_VRT_HME_FB THEN
	OP90_SRV_LH_VERT_CNTRL.ABSmove_Start	:= FALSE;
	OP90_A_SRV_LHVERT_HME					:= FALSE;
END_IF
END_IF

IF OP90_A_SRV_LHVERT_PCKWRK AND NOT OP90_A_SRV_LHVERT_HME AND NOT OP90_A_SRV_LHVERT_SPLCWRK AND NOT OP90_A_SRV_LHVERT_PLCWRK THEN
	OP90_SRV_LH_VERT_CNTRL.ABSmove_Start	:= TRUE;
	OP90_SRV_LH_VERT_CNTRL.Position			:= OP90_SRV_VERT_LH_PCKWRK_MM ;
IF OP90_SRV_LH_VRT_PCKWRK_FB THEN
	OP90_A_SRV_LHVERT_PCKWRK				:= FALSE;
	OP90_SRV_LH_VERT_CNTRL.ABSmove_Start	:= FALSE;
END_IF
END_IF

IF OP90_A_SRV_LHVERT_SPLCWRK AND NOT OP90_A_SRV_LHVERT_HME AND NOT OP90_A_SRV_LHVERT_PCKWRK AND NOT OP90_A_SRV_LHVERT_PLCWRK THEN
	OP90_SRV_LH_VERT_CNTRL.ABSmove_Start	:= TRUE;
	OP90_SRV_LH_VERT_CNTRL.Position			:= OP90_SRV_VERT_LH_SPLCWRK_MM ;
IF OP90_SRV_LH_VRT_SPLCWRK_FB THEN
	OP90_SRV_LH_VERT_CNTRL.ABSmove_Start	:= FALSE;
	OP90_A_SRV_LHVERT_SPLCWRK				:= FALSE;
END_IF
END_IF

IF OP90_A_SRV_LHVERT_PLCWRK AND NOT OP90_A_SRV_LHVERT_HME AND NOT OP90_A_SRV_LHVERT_PCKWRK AND NOT OP90_A_SRV_LHVERT_SPLCWRK THEN
	OP90_SRV_LH_VERT_CNTRL.ABSmove_Start	:= TRUE;
	OP90_SRV_LH_VERT_CNTRL.Position			:= OP90_SRV_VERT_LH_PLCWRK_MM ;
IF OP90_SRV_LH_VRT_PLCWRK_FB THEN
	OP90_SRV_LH_VERT_CNTRL.ABSmove_Start	:= FALSE;
	OP90_A_SRV_LHVERT_PLCWRK				:= FALSE;
END_IF
END_IF
//////////////////////////////////////OP90_RH VRT HMR WRK//////////////////////////////////////////////
IF OP90_A_SRV_RHVERT_HME AND NOT OP90_A_SRV_RHVERT_PCKWRK AND NOT OP90_A_SRV_RHVERT_SPLCWRK AND NOT OP90_A_SRV_RHVERT_PLCWRK THEN
	OP90_SRV_RH_VERT_CNTRL.ABSmove_Start	:= TRUE;
	OP90_SRV_RH_VERT_CNTRL.Position			:= OP90_SRV_VERT_RH_HME_MM ;
IF OP90_SRV_RH_VRT_HME_FB THEN
	OP90_SRV_RH_VERT_CNTRL.ABSmove_Start	:= FALSE;
	OP90_A_SRV_RHVERT_HME					:= FALSE;
END_IF
END_IF

IF OP90_A_SRV_RHVERT_PCKWRK AND NOT OP90_A_SRV_RHVERT_HME AND NOT OP90_A_SRV_RHVERT_SPLCWRK AND NOT OP90_A_SRV_RHVERT_PLCWRK THEN
	OP90_SRV_RH_VERT_CNTRL.ABSmove_Start	:= TRUE;
	OP90_SRV_RH_VERT_CNTRL.Position			:= OP90_SRV_VERT_RH_PCKWRK_MM ;
IF OP90_SRV_RH_VRT_PCKWRK_FB THEN
	OP90_SRV_RH_VERT_CNTRL.ABSmove_Start	:= FALSE;
	OP90_A_SRV_RHVERT_PCKWRK				:= FALSE;
END_IF
END_IF

IF OP90_A_SRV_RHVERT_SPLCWRK AND NOT OP90_A_SRV_RHVERT_HME AND NOT OP90_A_SRV_RHVERT_PCKWRK AND NOT OP90_A_SRV_RHVERT_PLCWRK THEN
	OP90_SRV_RH_VERT_CNTRL.ABSmove_Start	:= TRUE;
	OP90_SRV_RH_VERT_CNTRL.Position			:= OP90_SRV_VERT_RH_SPLCWRK_MM ;
IF OP90_SRV_RH_VRT_SPLCWRK_FB THEN
	OP90_SRV_RH_VERT_CNTRL.ABSmove_Start	:= FALSE;
	OP90_A_SRV_RHVERT_SPLCWRK				:= FALSE;
END_IF
END_IF

IF OP90_A_SRV_RHVERT_PLCWRK AND NOT OP90_A_SRV_RHVERT_HME AND NOT OP90_A_SRV_RHVERT_PCKWRK AND NOT OP90_A_SRV_RHVERT_SPLCWRK THEN
	OP90_SRV_RH_VERT_CNTRL.ABSmove_Start	:= TRUE;
	OP90_SRV_RH_VERT_CNTRL.Position			:= OP90_SRV_VERT_RH_PLCWRK_MM ;
IF OP90_SRV_RH_VRT_PLCWRK_FB THEN
	OP90_SRV_RH_VERT_CNTRL.ABSmove_Start	:= FALSE;
	OP90_A_SRV_RHVERT_PLCWRK				:= FALSE;
END_IF
END_IF

///////////////////////////////OP90 ROTARY STEPPER HME WRK///////////////////////////////////////////

IF OP90_A_SRV_LH_ROTRY_HME AND NOT OP90_A_SRV_LH_ROTRY_WRK THEN
	OP90_STP_LH_ROTRY_CNTRL.ABSmove_Start	:= TRUE;
	OP90_STP_LH_ROTRY_CNTRL.Position		:= OP90_STP_ROTRY_LH_HME_MM;
IF OP90_STP_LH_ROTY_HME_FB THEN
	OP90_STP_LH_ROTRY_CNTRL.ABSmove_Start	:= FALSE;
	OP90_A_SRV_LH_ROTRY_HME					:= FALSE;
END_IF
END_IF

IF OP90_A_SRV_LH_ROTRY_WRK AND NOT OP90_A_SRV_LH_ROTRY_HME THEN
	OP90_STP_LH_ROTRY_CNTRL.ABSmove_Start	:= TRUE;
	OP90_STP_LH_ROTRY_CNTRL.Position		:= OP90_STP_ROTRY_LH_WRK_MM;
IF OP90_STP_LH_ROTY_WRK_FB THEN
	OP90_STP_LH_ROTRY_CNTRL.ABSmove_Start	:= FALSE;
	OP90_A_SRV_LH_ROTRY_WRK					:= FALSE;
END_IF
END_IF

IF OP90_A_SRV_RH_ROTRY_HME AND NOT OP90_A_SRV_RH_ROTRY_WRK THEN
	OP90_STP_RH_ROTRY_CNTRL.ABSmove_Start	:= TRUE;
	OP90_STP_RH_ROTRY_CNTRL.Position		:= OP90_STP_ROTRY_RH_HME_MM;
IF OP90_STP_RH_ROTY_HME_FB THEN
	OP90_STP_RH_ROTRY_CNTRL.ABSmove_Start	:= FALSE;
	OP90_A_SRV_RH_ROTRY_HME					:= FALSE;
END_IF
END_IF

IF OP90_A_SRV_RH_ROTRY_WRK AND NOT OP90_A_SRV_RH_ROTRY_HME THEN
	OP90_STP_RH_ROTRY_CNTRL.ABSmove_Start	:= TRUE;
	OP90_STP_RH_ROTRY_CNTRL.Position		:= OP90_STP_ROTRY_RH_WRK_MM;
IF OP90_STP_RH_ROTY_WRK_FB THEN
	OP90_STP_RH_ROTRY_CNTRL.ABSmove_Start	:= FALSE;
	OP90_A_SRV_RH_ROTRY_WRK					:= FALSE;
END_IF
END_IF


// FEEDBACK CONDITION

OP90_SRV_HORZ_HME_FB					:= OP90_SRV_HORZ_CNTRL.Axis_In_Pos AND In_Range(value:=OP90_SRV_HORZ_STATUS.actualPosition, setvalue:=OP90_SRV_HORZ_HME_MM , tolerance:=0.2 );
OP90_SRV_HORZ_ZERO_FB					:= OP90_SRV_HORZ_CNTRL.Axis_In_Pos AND In_Range(value:=OP90_SRV_HORZ_STATUS.actualPosition, setvalue:=0, tolerance:=0.2 );
OP90_SRV_HORZ_WRK_FB                    := OP90_SRV_HORZ_CNTRL.Axis_In_Pos AND In_Range(value:=OP90_SRV_HORZ_STATUS.actualPosition, setvalue:=OP90_SRV_HORZ_WRK_MM , tolerance:=0.2 );
OP90_SRV_LH_VRT_HME_FB                  := OP90_SRV_LH_VERT_CNTRL.Axis_In_Pos AND In_Range(value:=OP90_SRV_LH_VERT_STATUS.actualPosition, setvalue:=OP90_SRV_VERT_LH_HME_MM , tolerance:=0.2 );
OP90_SRV_LH_VRT_ZERO_FB                 := OP90_SRV_LH_VERT_CNTRL.Axis_In_Pos AND In_Range(value:=OP90_SRV_LH_VERT_STATUS.actualPosition, setvalue:=0, tolerance:=0.2 );
OP90_SRV_RH_VRT_HME_FB                  := OP90_SRV_RH_VERT_CNTRL.Axis_In_Pos AND In_Range(value:=OP90_SRV_RH_VERT_STATUS.actualPosition, setvalue:=OP90_SRV_VERT_RH_HME_MM , tolerance:=0.2 );
OP90_SRV_RH_VRT_ZERO_FB                 := OP90_SRV_RH_VERT_CNTRL.Axis_In_Pos AND In_Range(value:=OP90_SRV_RH_VERT_STATUS.actualPosition, setvalue:=0, tolerance:=0.2 );
OP90_SRV_LH_VRT_PCKWRK_FB               := OP90_SRV_LH_VERT_CNTRL.Axis_In_Pos AND In_Range(value:=OP90_SRV_LH_VERT_STATUS.actualPosition, setvalue:=OP90_SRV_VERT_LH_PCKWRK_MM , tolerance:=0.2 );
OP90_SRV_RH_VRT_PCKWRK_FB               := OP90_SRV_RH_VERT_CNTRL.Axis_In_Pos AND In_Range(value:=OP90_SRV_RH_VERT_STATUS.actualPosition, setvalue:=OP90_SRV_VERT_RH_PCKWRK_MM , tolerance:=0.2 );
OP90_SRV_LH_VRT_SPLCWRK_FB              := OP90_SRV_LH_VERT_CNTRL.Axis_In_Pos AND In_Range(value:=OP90_SRV_LH_VERT_STATUS.actualPosition, setvalue:=OP90_SRV_VERT_LH_SPLCWRK_MM , tolerance:=0.2 );
OP90_SRV_RH_VRT_SPLCWRK_FB              := OP90_SRV_RH_VERT_CNTRL.Axis_In_Pos AND In_Range(value:=OP90_SRV_RH_VERT_STATUS.actualPosition, setvalue:=OP90_SRV_VERT_RH_SPLCWRK_MM , tolerance:=0.2 );
OP90_SRV_LH_VRT_PLCWRK_FB               := OP90_SRV_LH_VERT_CNTRL.Axis_In_Pos AND In_Range(value:=OP90_SRV_LH_VERT_STATUS.actualPosition, setvalue:=OP90_SRV_VERT_LH_PLCWRK_MM , tolerance:=0.2 );
OP90_SRV_RH_VRT_PLCWRK_FB               := OP90_SRV_RH_VERT_CNTRL.Axis_In_Pos AND In_Range(value:=OP90_SRV_RH_VERT_STATUS.actualPosition, setvalue:=OP90_SRV_VERT_RH_PLCWRK_MM , tolerance:=0.2 );
OP90_STP_LH_ROTY_HME_FB					:= OP90_STP_LH_ROTRY_CNTRL.Axis_In_Pos AND In_Range(value:=OP90_STP_LH_ROTRY_STATUS.actualPosition, setvalue:=OP90_STP_ROTRY_LH_HME_MM , tolerance:=0.2 );;
OP90_STP_LH_ROTY_WRK_FB					:= OP90_STP_LH_ROTRY_CNTRL.Axis_In_Pos AND In_Range(value:=OP90_STP_LH_ROTRY_STATUS.actualPosition, setvalue:=OP90_STP_ROTRY_LH_WRK_MM , tolerance:=0.2 );; 
OP90_STP_RH_ROTY_HME_FB                 := OP90_STP_RH_ROTRY_CNTRL.Axis_In_Pos AND In_Range(value:=OP90_STP_RH_ROTRY_STATUS.actualPosition, setvalue:=OP90_STP_ROTRY_RH_HME_MM , tolerance:=0.2 );; 
OP90_STP_RH_ROTY_WRK_FB                 := OP90_STP_RH_ROTRY_CNTRL.Axis_In_Pos AND In_Range(value:=OP90_STP_RH_ROTRY_STATUS.actualPosition, setvalue:=OP90_STP_ROTRY_RH_WRK_MM , tolerance:=0.2 );; 
OP90_VERT_SRV_SAFE_ZONE					:=(OP90_SRV_VERT_LH_HME_MM<OP90_SRV_LH_VERT_STATUS.actualPosition AND OP90_SRV_LH_VERT_STATUS.actualPosition<OP90_SRV_VERT_LH_SPLCWRK_MM AND 
											OP90_SRV_VERT_RH_HME_MM<OP90_SRV_RH_VERT_STATUS.actualPosition AND OP90_SRV_RH_VERT_STATUS.actualPosition<OP90_SRV_VERT_RH_SPLCWRK_MM ); 	

                                           
////////////////////////////FUNCTIONAL BLOCK/////////////////////////////

OP90_SRV_HORZ(
	bAxis1_Ref_Switch:= , 
	bInit:= OP90_BLCK_INITZ, 
	bErrorReset:= Servo_Reset , 														// ERROR RESET
	bEnable:= Servo_Enable,
	bMoveVelocity:= , 
	bHalt:= , 
	bManualMode:= OP90_MANUAL_SELECTED, 
	fHomePos:= , 
	fOverride:= , 
	fTargetPosition:= OP90_SRV_HORZ_CNTRL.Position, 
	fTargetVelocity:= OP90_SRV_LIMIT.OP90_A_HORZ_VELOCITY,
	fAcc:= , 
	fDec:= ,
	Servo_High_Limit:=OP90_SRV_LIMIT.OP90_HORZ_POS_LIMIT,	
	Servo_Low_Limit:=OP90_SRV_LIMIT.OP90_HORZ_NEG_LIMIT,	 	
	WARNING_LIMIT:=1, 
	Safe_move_Conditions:=Servo_Safety,
	TORQUE_APPLIED := , 
	Axis:= OP90_SRVO_HORZ, 
	bHome:= OP90_SRV_HORZ_CNTRL.Axis_Home_Cmd, 
	bSetPosition:= FESTO_NOT_NEED , 
	bMoveAbsolute:= OP90_SRV_HORZ_CNTRL.ABSmove_Start, 
	bMoveRelative:= NOT_REF , 
	bMoveTorque:= NOT_REF , 
	stManualModeAxis:= OP90_SRV_HORZ_STATUS, 
	sAxisState=>OP90_SRV_HORZ_FB, 
	bAxis_ready=> , 
	bAxisInPosition=> , 
	bAxisError=> , 
	bAxisEnabled=> , 
	bAxisHomed=> OP90_SRV_HORZ_CNTRL.Axis_reference, 
	bSetPositionDone=> , 
	bHaltDone=> , 
	bSTOPDone=> , 
	bHomeDone=> , 
	bDone=> , 
	bTorqueReached=> , 
	bsafe_to_move=> , 
	baxis_in_home_pos=> , 
	bABS_Pos_done=> OP90_SRV_HORZ_CNTRL.Axis_In_Pos, 
	Actual_position=> , 
	Actual_velocity=> , 
	Actual_Torque=> );
	
OP90_SRV_LH_VERT(
	bAxis1_Ref_Switch:= , 
	bInit:=  OP90_BLCK_INITZ, 
	bErrorReset:= Servo_Reset, 
	bEnable:= Servo_Enable, 
	bMoveVelocity:= , 
	bHalt:= , 
	bManualMode:= OP90_MANUAL_SELECTED, 
	fHomePos:= , 
	fOverride:= , 
	fTargetPosition:= OP90_SRV_LH_VERT_CNTRL.Position	, 
	fTargetVelocity:= OP90_SRV_LIMIT.OP90_A_LH_VERT_VELOCITY, 
	fAcc:= , 
	fDec:= ,
	Servo_High_Limit:= OP90_SRV_LIMIT.OP90_LH_VERT_POS_LIMIT,	
	Servo_Low_Limit:=OP90_SRV_LIMIT.OP90_LH_VERT_NEG_LIMIT,	 	
	WARNING_LIMIT:=1, 
	Safe_move_Conditions:=Servo_Safety,
	TORQUE_APPLIED := , 
	Axis:= OP90_SRVO_LH_VERT, 
	bHome:= OP90_SRV_LH_VERT_CNTRL.Axis_Home_Cmd, 
	bSetPosition:= FESTO_NOT_NEED , 
	bMoveAbsolute:= OP90_SRV_LH_VERT_CNTRL.ABSmove_Start, 
	bMoveRelative:= NOT_REF , 
	bMoveTorque:= NOT_REF , 
	stManualModeAxis:= OP90_SRV_LH_VERT_STATUS, 
	sAxisState=> OP90_SRV_LH_VERT_FB, 
	bAxis_ready=> , 
	bAxisInPosition=>, 
	bAxisError=> , 
	bAxisEnabled=> , 
	bAxisHomed=>OP90_SRV_LH_VERT_CNTRL.Axis_reference, 
	bSetPositionDone=> , 
	bHaltDone=> , 
	bSTOPDone=> , 
	bHomeDone=> , 
	bDone=> , 
	bTorqueReached=> , 
	bsafe_to_move=> , 
	baxis_in_home_pos=> , 
	bABS_Pos_done=>  OP90_SRV_LH_VERT_CNTRL.Axis_In_Pos, 
	Actual_position=> , 
	Actual_velocity=> , 
	Actual_Torque=> OP90_SRV_LH_VERT_CNTRL.Actual_Torque);
	
	
OP90_SRV_RH_VERT(
	bAxis1_Ref_Switch:= , 
	bInit:=  OP90_BLCK_INITZ, 
	bErrorReset:= Servo_Reset, 
	bEnable:= Servo_Enable, 
	bMoveVelocity:= , 
	bHalt:= , 
	bManualMode:=OP90_MANUAL_SELECTED , 
	fHomePos:= , 
	fOverride:= , 
	fTargetPosition:= OP90_SRV_RH_VERT_CNTRL.Position, 
	fTargetVelocity:= OP90_SRV_LIMIT.OP90_A_RH_VERT_VELOCITY, 
	fAcc:= , 
	fDec:= ,
	Servo_High_Limit:= OP90_SRV_LIMIT.OP90_RH_VERT_POS_LIMIT,	
	Servo_Low_Limit:=OP90_SRV_LIMIT.OP90_RH_VERT_NEG_LIMIT,	 	
	WARNING_LIMIT:=1, 
	Safe_move_Conditions:=Servo_Safety,
	TORQUE_APPLIED :=  , 
	Axis:= OP90_SRVO_RH_VERT, 
	bHome:= OP90_SRV_RH_VERT_CNTRL.Axis_Home_Cmd, 
	bSetPosition:= FESTO_NOT_NEED , 
	bMoveAbsolute:= OP90_SRV_RH_VERT_CNTRL.ABSmove_Start, 
	bMoveRelative:= NOT_REF , 
	bMoveTorque:= NOT_REF , 
	stManualModeAxis:= OP90_SRV_RH_VERT_STATUS, 
	sAxisState=> OP90_SRV_RH_VERT_FB, 
	bAxis_ready=> , 
	bAxisInPosition=> , 
	bAxisError=> , 
	bAxisEnabled=> , 
	bAxisHomed=>OP90_SRV_RH_VERT_CNTRL.Axis_reference, 
	bSetPositionDone=> , 
	bHaltDone=> , 
	bSTOPDone=> , 
	bHomeDone=> , 
	bDone=> , 
	bTorqueReached=> , 
	bsafe_to_move=> , 
	baxis_in_home_pos=> , 
	bABS_Pos_done=> OP90_SRV_RH_VERT_CNTRL.Axis_In_Pos, 
	Actual_position=> , 
	Actual_velocity=> , 
	Actual_Torque=> );	
	
OP90_GUIDE_SERVO(
	bAxis1_Ref_Switch:= , 
	bInit:= OP90_BLCK_INITZ, 
	bErrorReset:= Servo_Reset, 
	bEnable:= Servo_Enable, 
	bMoveVelocity:= , 
	bHalt:= , 
	bManualMode:=OP90_MANUAL_SELECTED, 
	fHomePos:= , 
	fOverride:= , 
	fTargetPosition:= OP90_SERVO_GUIDE_CNTRL.Position, 
	fTargetVelocity:= OP90_SERVO_GUIDE_CNTRL.Velocity, 
	fAcc:= , 
	fDec:= ,
	Servo_High_Limit:= OP90_SRV_LIMIT.OP90_GUIDE_POS_LIMIT,	
	Servo_Low_Limit:=OP90_SRV_LIMIT.OP90_GUIDE_NEG_LIMIT,	 	
	WARNING_LIMIT:=1, 
	Safe_move_Conditions:= Servo_Safety,
	TORQUE_APPLIED := , 
	Axis:= OP90_GUID_SERV, 
	bHome:= OP90_SERVO_GUIDE_CNTRL.Axis_Home_Cmd, 
	bSetPosition:= FESTO_NOT_NEED, 
	bMoveAbsolute:= OP90_SERVO_GUIDE_CNTRL.ABSmove_Start, 
	bMoveRelative:= NOT_REF, 
	bMoveTorque:= NOT_REF, 
	stManualModeAxis:= OP90_GIUDE_SER_STATUS, 
	sAxisState=> OP90_SRV_GUID_STOPER_FB, 
	bAxis_ready=>OP90_SERVO_GUIDE_CNTRL.Axis_ready , 
	bAxisInPosition=> , 
	bAxisError=> , 
	bAxisEnabled=> , 
	bAxisHomed=> OP90_SERVO_GUIDE_CNTRL.Axis_reference, 
	bSetPositionDone=> , 
	bHaltDone=> , 
	bSTOPDone=> , 
	bHomeDone=> , 
	bDone=> , 
	bTorqueReached=> , 
	bsafe_to_move=> , 
	baxis_in_home_pos=> , 
	bABS_Pos_done=> OP90_SERVO_GUIDE_CNTRL.Axis_In_Pos, 
	Actual_position=>OP90_SERVO_GUIDE_CNTRL.Actual_Position , 
	Actual_velocity=>OP90_SERVO_GUIDE_CNTRL.Actual_Velocity , 
	Actual_Torque=> );
	
OP90_LH_SRV_ROTRY(
	bAxis1_Ref_Switch:= , 
	bInit:= OP90_BLCK_INITZ, 
	bErrorReset:= Servo_Reset, 
	bEnable:= Servo_Enable, 
	bMoveVelocity:= , 
	bHalt:= , 
	bManualMode:=OP90_MANUAL_SELECTED, 
	fHomePos:= , 
	fOverride:= , 
	fTargetPosition:= OP90_STP_LH_ROTRY_CNTRL.Position, 
	fTargetVelocity:= OP90_SRV_LIMIT.OP90_A_LH_ROTRY_VELOCITY, 
	fAcc:= , 
	fDec:= ,
	Servo_High_Limit:= OP90_SRV_LIMIT.OP90_LH_ROTRY_POS_LIMIT,	
	Servo_Low_Limit:=OP90_SRV_LIMIT.OP90_LH_ROTRY_NEG_LIMIT,	 	
	WARNING_LIMIT:=1, 
	Safe_move_Conditions:= Servo_Safety,
	TORQUE_APPLIED := , 
	Axis:= OP90_STP_LH_ROTRY, 
	bHome:= OP90_STP_LH_ROTRY_CNTRL.Axis_Home_Cmd, 
	bSetPosition:= FESTO_NOT_NEED, 
	bMoveAbsolute:= OP90_STP_LH_ROTRY_CNTRL.ABSmove_Start, 
	bMoveRelative:= NOT_REF, 
	bMoveTorque:= NOT_REF, 
	stManualModeAxis:= OP90_STP_LH_ROTRY_STATUS, 
	sAxisState=> OP90_LH_ROTARY_STUTS, 
	bAxis_ready=> , 
	bAxisInPosition=>, 
	bAxisError=> , 
	bAxisEnabled=> , 
	bAxisHomed=> OP90_STP_LH_ROTRY_CNTRL.Axis_reference, 
	bSetPositionDone=> , 
	bHaltDone=> , 
	bSTOPDone=> , 
	bHomeDone=> , 
	bDone=> , 
	bTorqueReached=> , 
	bsafe_to_move=> , 
	baxis_in_home_pos=> , 
	bABS_Pos_done=> OP90_STP_LH_ROTRY_CNTRL.Axis_In_Pos, 
	Actual_position=> , 
	Actual_velocity=> , 
	Actual_Torque=> );
	
	
OP90_RH_SRV_ROTRY(
	bAxis1_Ref_Switch:= , 
	bInit:= OP90_BLCK_INITZ, 
	bErrorReset:=Servo_Reset, 
	bEnable:= Servo_Enable, 
	bMoveVelocity:= , 
	bHalt:= , 
	bManualMode:=OP90_MANUAL_SELECTED, 
	fHomePos:= , 
	fOverride:= , 
	fTargetPosition:= OP90_STP_RH_ROTRY_CNTRL.Position, 
	fTargetVelocity:= OP90_SRV_LIMIT.OP90_A_RH_ROTRY_VELOCITY, 
	fAcc:= , 
	fDec:= ,
	Servo_High_Limit:= OP90_SRV_LIMIT.OP90_RH_ROTRY_POS_LIMIT,	
	Servo_Low_Limit:=OP90_SRV_LIMIT.OP90_RH_ROTRY_NEG_LIMIT,	 	
	WARNING_LIMIT:=1, 
	Safe_move_Conditions:= Servo_Safety,
	TORQUE_APPLIED := , 
	Axis:= OP90_STP_RH_ROTRY, 
	bHome:= OP90_STP_RH_ROTRY_CNTRL.Axis_Home_Cmd, 
	bSetPosition:= FESTO_NOT_NEED, 
	bMoveAbsolute:= OP90_STP_RH_ROTRY_CNTRL.ABSmove_Start, 
	bMoveRelative:= NOT_REF, 
	bMoveTorque:= NOT_REF, 
	stManualModeAxis:= OP90_STP_RH_ROTRY_STATUS, 
	sAxisState=> OP90_RH_ROTARY_STUTS, 
	bAxis_ready=> , 
	bAxisInPosition=>, 
	bAxisError=> , 
	bAxisEnabled=> , 
	bAxisHomed=> OP90_STP_RH_ROTRY_CNTRL.Axis_reference, 
	bSetPositionDone=> , 
	bHaltDone=> , 
	bSTOPDone=> , 
	bHomeDone=> , 
	bDone=> , 
	bTorqueReached=> , 
	bsafe_to_move=> , 
	baxis_in_home_pos=> , 
	bABS_Pos_done=> OP90_STP_RH_ROTRY_CNTRL.Axis_In_Pos, 
	Actual_position=> , 
	Actual_velocity=> , 
	Actual_Torque=> );	
	


OP90_LH_CNVY(
	bAxis1_Ref_Switch:= , 
	bInit:= , 
	bErrorReset:= Servo_Reset, 
	bEnable:= Servo_Enable, 
	bMoveVelocity:=OP90_SRV_LH_CNVY_CNTRL.VELmove_Start , 
	bHalt:= , 
	bManualMode:=OP90_MANUAL_SELECTED, 
	fHomePos:= , 
	fOverride:= , 
	fTargetPosition:=OP90_SRV_LH_CNVY_CNTRL.Position , 
	fTargetVelocity:=OP90_SRV_LH_CNVY_CNTRL.Velocity , 
	fAcc:= , 
	fDec:= ,
	LIMIT_BYPASS:=1, 
	Servo_High_Limit:= 50,	
	Servo_Low_Limit:=0,	 	
	WARNING_LIMIT:=1, 
	Safe_move_Conditions:=Servo_Safety , 
	Axis:= OP90_SRV_CNVY_RH, 
	HME_WRITE_ADD:= 16#5010,	
	bHome:= OP90_SRV_LH_CNVY_CNTRL.Bsethome, 
	bSetPosition:= OP90_SRV_LH_CNVY_CNTRL.BsetPos ,
	bMoveVelocity:=OP90_SRV_LH_CNVY_CNTRL.VELmove_Start , 
	bMoveAbsolute:=OP90_SRV_LH_CNVY_CNTRL.ABSmove_Start , 
	bMoveRelative:=OP90_SRV_LH_CNVY_CNTRL.RELmove_Start, 
	bMoveTorque:= OP90_SRV_LH_CNVY_CNTRL.Torque_mode_Start, 
	stManualModeAxis:= OP90_SRV_LH_CNVY_STATUS, 
	bmove_home:=OP90_SRV_LH_CNVY_CNTRL.Axis_Home_Cmd , 
	sAxisState=> OP90_SRV_LH_CNVY_CNTRL.Axis_State, 
	bAxis_ready=>OP90_SRV_LH_CNVY_CNTRL.Axis_ready , 
	bAxisInPosition=> , 
	bAxisError=> OP90_SRV_LH_CNVY_CNTRL.Axis_Error, 
	bAxisEnabled=> , 
	bAxisHomed=> OP90_SRV_LH_CNVY_CNTRL.Axis_reference, 
	bSetPositionDone=> , 
	bHaltDone=> , 
	bSTOPDone=> , 
	bHomeDone=> , 
	bDone=> , 
	bTorqueReached=> , 
	bsafe_to_move=> , 
	baxis_in_home_pos=> , 
	bABS_Pos_done=> , 
	Actual_position=> , 
	Actual_velocity=> , 
	Actual_Torque=> );	
	
OP90_RH_CNVY(
    bAxis1_Ref_Switch:= , 
	bInit:= , 
	bErrorReset:= Servo_Reset, 
	bEnable:= Servo_Enable, 
	bHalt:= , 
	bManualMode:= OP90_MANUAL_SELECTED, 
	fHomePos:= , 
	fOverride:= , 
	fTargetPosition:= OP90_SRV_RH_CNVY_CNTRL.Position, 
	fTargetVelocity:= OP90_SRV_RH_CNVY_CNTRL.Velocity, 
	fAcc:= , 
	fDec:= ,
	LIMIT_BYPASS:=1, 
	Servo_High_Limit:= 50,	
	Servo_Low_Limit:=0,	 	
	WARNING_LIMIT:=1, 
	Safe_move_Conditions:=Servo_Safety, 
	Axis:= OP90_SRV_CNVY_LH, 
	HME_WRITE_ADD:= 16#5011,	
	bHome:= OP90_SRV_RH_CNVY_CNTRL.Bsethome, 
	bSetPosition:= OP90_SRV_RH_CNVY_CNTRL.BsetPos ,
	bMoveVelocity:=OP90_SRV_RH_CNVY_CNTRL.VELmove_Start , 
	bMoveAbsolute:=OP90_SRV_RH_CNVY_CNTRL.ABSmove_Start , 
	bMoveRelative:=OP90_SRV_RH_CNVY_CNTRL.RELmove_Start, 
	bMoveTorque:= OP90_SRV_RH_CNVY_CNTRL.Torque_mode_Start, 
	stManualModeAxis:= OP90_SRV_RH_CNVY_STATUS, 
	bmove_home:=OP90_SRV_RH_CNVY_CNTRL.Axis_Home_Cmd , 
	sAxisState=>OP90_SRV_RH_CNVY_CNTRL.Axis_State , 
	bAxis_ready=>OP90_SRV_RH_CNVY_CNTRL.Axis_ready , 
	bAxisInPosition=> , 
	bAxisError=> OP90_SRV_RH_CNVY_CNTRL.Axis_Error, 
	bAxisEnabled=> , 
	bAxisHomed=> OP90_SRV_RH_CNVY_CNTRL.Axis_reference, 
	bSetPositionDone=> , 
	bHaltDone=> , 
	bSTOPDone=> , 
	bHomeDone=> , 
	bDone=> , 
	bTorqueReached=> , 
	bsafe_to_move=> , 
	baxis_in_home_pos=> , 
	bABS_Pos_done=> , 
	Actual_position=> , 
	Actual_velocity=> , 
	Actual_Torque=> );
	
IF OP90_MANUAL_SELECTED THEN
	OP90_SRV_HORZ_STATUS.targetVelocity:=50;
	OP90_SRV_LH_VERT_STATUS.targetVelocity:=50;
	OP90_SRV_RH_VERT_STATUS.targetVelocity:=50;
	OP90_STP_LH_ROTRY_STATUS.targetVelocity:=50;
	OP90_STP_RH_ROTRY_STATUS.targetVelocity:=50;
	OP90_GIUDE_SER_STATUS.targetVelocity:=50;
	//OP90_SRV_LH_CNVY_STATUS.targetVelocity:=100;
	//OP90_SRV_RH_CNVY_STATUS.targetVelocity:=100; 	
END_IF

END_PROGRAM

// ---- POUs/Programs/OP90/OP90_AUTO.TcPOU
PROGRAM OP90_AUTO
VAR
	
// TON
	AFT_SUP_HRZ_WRK				: TON;
	AFT_VERT_PCK_WRK			: TON;
	AFT_PCK_DN					: TON;
	AFT_VRT_PLC_WRK				: TON;
	AFT_GRP_HME					: TON;
	AFT_VRT_SUP_HME				: TON;
	AFT_SUP_CYL_HME				: TON;
//INT
	OP90_STP_NO					: INT;
//BOOL

	OP90_LH_CMP_OK				: BOOL;
	OP90_RH_CMP_OK				: BOOL;
	

	OP90_STN_MOVER: INT;

	Track_1_TMR : TON;
	Track_2_TMR : TON;
	Track_3_TMR : TON;
	Track_4_TMR : TON;
	Track_5_TMR : TON;
	Track_6_TMR : TON;
	Track_7_TMR : TON;
	Track_8_TMR : TON;
	Track_9_TMR : TON;
	Track_10_TMR : TON;
	Track_11_TMR : TON;
	Track_12_TMR : TON;	
	
	
	
	dllky: Ton;
	OP90_RH_CMP_TORQE_OK: BOOL;
	OP90_LH_CMP_TORQE_OK: BOOL;
END_VAR

VAR PERSISTENT
	OP90_Auto_Status			: STRING;
	OP90_AFT_SUP_HRZ_WRK		: INT;
	OP90_AFT_VRT_PCK_WRK		: INT;
	OP90_AFT_CMP_PCK			: INT;
	OP90_AFT_VRT_PLC_WRK		: INT;
	OP90_AFT_GRP_HME			: INT;
	OP90_AFT_SUP_VRT_HME		: INT;
	OP90_AFT_SUP_CYL_HME		: INT;
	OP90_Guide_Servo_Position   : REAL := 73;
END_VAR

///////Status message///////////

IF OP90_STP_NO=0 AND NOT OP90_ALL_HOME THEN
	OP90_Auto_Status:='Homing not Done';
ELSIF  OP90_STP_NO=0 AND OP90_ALL_HOME THEN
	OP90_Auto_Status:='Press Cycle Start';
ELSIF  OP90_STP_NO=1 AND ((OP90_LH_CMP_PICKED AND OP90_RH_CMP_PICKED) OR OP90_pick_ready)  THEN
	OP90_Auto_Status:='Component Picked';	
ELSIF  OP90_STP_NO=1 AND NOT OP90_pick_ready THEN
	OP90_Auto_Status:='Waiting For Conveyor Singulation';
ELSIF  OP90_STP_NO=5  THEN
	OP90_Auto_Status:='Horizontal Servo moving to Pick Position';
ELSIF  OP90_STP_NO=10  THEN
	OP90_Auto_Status:='Vertical Servo moving to Place Position';
ELSIF  OP90_STP_NO=15  THEN
	OP90_Auto_Status:='Waiting for Gripper Open Feedback';	
ELSIF  OP90_STP_NO=20  THEN
	OP90_Auto_Status:='Vertical Servo moving to Safe Position';	
ELSIF OP90_STP_NO=30  THEN
	OP90_Auto_Status:='Vertical Servo moving to Safe Place Position';	
ELSIF OP90_STP_NO=35  THEN
	OP90_Auto_Status:='Waiting Mover and Station Enable';	
ELSIF OP90_STP_NO=40  THEN
	OP90_Auto_Status:='Waiting for Gripper Close Feedback';	
ELSIF OP90_STP_NO=45  THEN
	OP90_Auto_Status:='Updating Result and Moving to next Cycle';
ELSIF OP90_STP_NO=50  THEN
	OP90_Auto_Status:='Vertical Servo moving to Safe Position';	
ELSIF OP90_STP_NO=55  THEN
	OP90_Auto_Status:='Supporting Cyclinder moving home';			
END_IF

IF OP90_AUTO_SELECTED OR OP90_STEP_SELECTED THEN
	OP90_SERVO_GUIDE_CNTRL.Position:=OP90_Guide_Servo_Position;
	OP90_SERVO_GUIDE_CNTRL.Velocity:=50;
ELSIF NOT (OP90_AUTO_RUNNING OR OP90_STEP_RUNNING) AND NOT In_Range(OP90_SERVO_GUIDE_CNTRL.Actual_Position,0,1) THEN
	OP90_SERVO_GUIDE_CNTRL.Position:=0;
	OP90_SERVO_GUIDE_CNTRL.Velocity:=50;
	OP90_SERVO_GUIDE_CNTRL.ABSmove_Start:=TRUE;
END_IF

IF OP90_AUTO_RUNNING OR OP90_STEP_RUNNING THEN

IF OP90_START_ENABLE THEN

IF OP90_STRT_PB AND OP90_ALL_HOME AND OP90_STP_NO=0 THEN
	OP90_SERVO_GUIDE_CNTRL.ABSmove_Start:=TRUE;
	OP90_STP_NO							:= 1;
END_IF

CASE OP90_STP_NO OF 
	1:	IF OP90_LH_CMP_PICKED AND OP90_RH_CMP_PICKED THEN
		OP90_STP_NO						:= 30;							
		ELSIF OP90_pick_ready THEN
		OP90_A_SRV_HORZ_WRK				:= TRUE;
		OP90_STP_NO						:= 5;		
		END_IF
	
	5:IF (OP90_LH_CMR_OK OR OP90_LH_CMP_PICKED) AND (OP90_RH_CMR_OK OR OP90_RH_CMP_PICKED) AND OP90_SRV_HORZ_WRK_FB THEN
		OP90_STP_NO						:= 10;	   
	   END_IF

	10: IF OP90_LH_CMP_PICKED AND NOT OP90_RH_CMP_PICKED  THEN
		OP90_A_SRV_LHVERT_PCKWRK		:= FALSE;
		OP90_A_SRV_RHVERT_PCKWRK 		:= TRUE;
		OP90_STP_NO						:= 15;
		END_IF
		IF NOT OP90_LH_CMP_PICKED AND  OP90_RH_CMP_PICKED  THEN
		OP90_A_SRV_LHVERT_PCKWRK		:= TRUE;
		OP90_A_SRV_RHVERT_PCKWRK 		:= FALSE;
		OP90_STP_NO						:= 15;
		END_IF		
		IF NOT OP90_LH_CMP_PICKED AND NOT OP90_RH_CMP_PICKED THEN
		OP90_A_SRV_LHVERT_PCKWRK		:= TRUE;
		OP90_A_SRV_RHVERT_PCKWRK 		:= TRUE;
		OP90_STP_NO						:= 15;			
		END_IF
	   
	   
	15: IF OP90_LH_CMP_PICKED AND NOT OP90_RH_CMP_PICKED AND OP90_SRV_RH_VRT_PCKWRK_FB AND AFT_VERT_PCK_WRK.Q  THEN
		OP90_A_RH_GRP_AUTCMD2			:= TRUE;
		OP90_A_RH_GRP_AUTCMD1			:= FALSE;		
		OP90_STP_NO						:= 20;
		END_IF
		IF NOT OP90_LH_CMP_PICKED AND  OP90_RH_CMP_PICKED AND OP90_SRV_LH_VRT_PCKWRK_FB AND AFT_VERT_PCK_WRK.Q THEN
		OP90_A_LH_GRP_AUTCMD2			:= TRUE;
		OP90_A_LH_GRP_AUTCMD1		    := FALSE;
		OP90_STP_NO						:= 20;
		END_IF		
		IF NOT OP90_LH_CMP_PICKED AND NOT OP90_RH_CMP_PICKED AND OP90_SRV_LH_VRT_PCKWRK_FB AND OP90_SRV_RH_VRT_PCKWRK_FB AND AFT_VERT_PCK_WRK.Q THEN
		OP90_A_RH_GRP_AUTCMD2			:= TRUE;
		OP90_A_RH_GRP_AUTCMD1			:= FALSE;
		OP90_A_LH_GRP_AUTCMD2			:= TRUE;
		OP90_A_LH_GRP_AUTCMD1		    := FALSE;
		OP90_STP_NO						:= 20;			
		END_IF

	20: IF AFT_PCK_DN.Q THEN
		OP90_LH_CMP_PICKED              := TRUE;
		OP90_RH_CMP_PICKED				:= TRUE;
		OP90_A_SRV_LHVERT_HME			:= TRUE;
		OP90_A_SRV_RHVERT_HME			:= TRUE;
		OP90_STP_NO						:= 25;		
		END_IF
	   
	25: IF OP90_SRV_LH_VRT_HME_FB AND OP90_SRV_RH_VRT_HME_FB THEN
		OP90_A_SRV_HORZ_HME				:= TRUE;
		OP90_pick_done_7_89				:= OP90_POS2_V7_89;
		OP90_pick_done_6_38				:= OP90_POS1_V6_3;
		OP90_A_SRV_LH_ROTRY_WRK			:= TRUE;
		OP90_A_SRV_RH_ROTRY_WRK			:= TRUE;		
		OP90_STP_NO						:= 30;		
		END_IF
		
	30: IF OP90_SRV_HORZ_HME_FB THEN                     	
		IF NOT OP90_STN_ENABLE THEN  	
		OP90_A_SRV_LHVERT_SPLCWRK		:= TRUE;
		OP90_A_SRV_RHVERT_SPLCWRK		:= TRUE;
 		OP90_STP_NO						:= 35;		
		ELSIF OP90_STN_ENABLE AND ((OP90_POS1_V6_3 AND OP90_SUP_VERTP1_CYL.Sensor2 )OR(OP90_POS2_V7_89 AND OP90_SUP_VERTP2_CYL.Sensor2)) THEN
		IF OP90_LH_CMP_OK THEN
		OP90_A_SRV_LHVERT_PLCWRK		:= TRUE;	
		END_IF	                    	
		IF OP90_RH_CMP_OK THEN      	
		OP90_A_SRV_RHVERT_PLCWRK		:= TRUE;	
		END_IF
		 OP90_STP_NO					:= 40;
		END_IF
		END_IF
		
	35: IF OP90_STN_ENABLE AND OP90_SRV_LH_VRT_SPLCWRK_FB AND OP90_SRV_RH_VRT_SPLCWRK_FB AND 
			((OP90_POS1_V6_3 AND OP90_SUP_VERTP1_CYL.Sensor2 )OR(OP90_POS2_V7_89 AND OP90_SUP_VERTP2_CYL.Sensor2 )) THEN
		IF OP90_LH_CMP_OK THEN
		OP90_A_SRV_LHVERT_PLCWRK		:= TRUE;
		OP90_A_SRV_LHVERT_SPLCWRK		:= FALSE;	
		END_IF	                    	
		IF OP90_RH_CMP_OK THEN      	
		OP90_A_SRV_RHVERT_PLCWRK		:= TRUE;
		OP90_A_SRV_RHVERT_SPLCWRK		:= FALSE;	
		END_IF
 		OP90_STP_NO						:= 40;	
		END_IF
		
	40: OP90_CURR_MOVER					:= OP90_STN_MOVER;
		OP90_LH_CMP_TORQE_OK			:= TRUE;					// NEED TO BE CHANGED BASED ON TORQUE FB
		OP90_RH_CMP_TORQE_OK			:= TRUE;					// NEED TO BE CHANGED BASED ON TORQUE FB
		IF OP90_LH_CMP_OK AND NOT OP90_RH_CMP_OK AND OP90_SRV_LH_VRT_PLCWRK_FB AND AFT_VRT_PLC_WRK.Q THEN
		OP90_A_LH_GRP_AUTCMD2			:= FALSE;
		OP90_A_LH_GRP_AUTCMD1		    := TRUE;
		OP90_LH_CMP_PICKED				:= FALSE; 
 		OP90_STP_NO						:= 45;	
  		END_IF
		IF NOT OP90_LH_CMP_OK AND  OP90_RH_CMP_OK AND OP90_SRV_RH_VRT_PLCWRK_FB AND AFT_VRT_PLC_WRK.Q THEN
		OP90_A_RH_GRP_AUTCMD2			:= FALSE;
		OP90_A_RH_GRP_AUTCMD1		    := TRUE;
		OP90_RH_CMP_PICKED				:= FALSE;
 		OP90_STP_NO						:= 45;
  		END_IF
		IF OP90_LH_CMP_OK AND OP90_RH_CMP_OK AND OP90_SRV_LH_VRT_PLCWRK_FB AND OP90_SRV_RH_VRT_PLCWRK_FB AND AFT_VRT_PLC_WRK.Q THEN
		OP90_A_LH_GRP_AUTCMD2			:= FALSE;
		OP90_A_LH_GRP_AUTCMD1		    := TRUE;
		OP90_A_RH_GRP_AUTCMD2			:= FALSE;
		OP90_A_RH_GRP_AUTCMD1		    := TRUE;
		OP90_LH_CMP_PICKED				:= FALSE;
		OP90_RH_CMP_PICKED              := FALSE;
 		OP90_STP_NO						:= 45;			
		END_IF
	
		
	45: IF OP90_STN_MOVER>0 THEN
		MOVER_CMP_STATUS[OP90_CURR_MOVER][1]:=90;
		MOVER_CMP_STATUS[OP90_CURR_MOVER][2]:=90;	
		END_IF
		IF OP90_LH_CMP_TORQE_OK AND NOT OP90_RH_CMP_OK AND I90_RET_LH_GRIPR_CYL_CLSE_I1200_0 THEN
		MOVER_CMP_STATUS[OP90_CURR_MOVER][1]:=90;
		MOVER_CMP_STATUS[OP90_CURR_MOVER][2]:=90;																////////////////////////////WRITE XTS AS OK/////////////////////////////																	
 		OP90_STP_NO						:= 50;		
		END_IF
		IF NOT OP90_LH_CMP_OK AND  OP90_RH_CMP_OK AND I90_RET_RH_GRIPR_CYL_CLSE_I1200_2 THEN
		MOVER_CMP_STATUS[OP90_CURR_MOVER][1]:=90;
		MOVER_CMP_STATUS[OP90_CURR_MOVER][2]:=90;																////////////////////////////WRITE XTS AS OK/////////////////////////////
 		OP90_STP_NO						:= 50;			
		END_IF
		IF OP90_LH_CMP_OK AND OP90_RH_CMP_OK AND I90_RET_LH_GRIPR_CYL_CLSE_I1200_0 AND I90_RET_RH_GRIPR_CYL_CLSE_I1200_2 THEN
																////////////////////////////WRITE XTS AS OK/////////////////////////////
 		OP90_STP_NO						:= 50;			
		END_IF
		
	50: IF AFT_GRP_HME.Q THEN
		OP90_A_SRV_LHVERT_HME			:= TRUE;
		OP90_A_SRV_RHVERT_HME			:= TRUE;
		OP90_A_MVR_SUP_VERTP1_HME		:= TRUE;
		OP90_A_MVR_SUP_VERTP1_WRK		:= FALSE;
		OP90_A_MVR_SUP_VERTP2_HME		:= TRUE;
		OP90_A_MVR_SUP_VERTP2_WRK		:= FALSE;
	   
		OP90_STP_NO						:= 55;
		END_IF			

	55: IF AFT_VRT_SUP_HME.Q THEN
		OP90_A_MVR_SUP_HORZP1_HME		:= TRUE;
		OP90_A_MVR_SUP_HORZP1_WRK		:= FALSE;
		OP90_A_MVR_SUP_HORZP2_HME		:= TRUE;
		OP90_A_MVR_SUP_HORZP2_WRK		:= FALSE;
 		OP90_STP_NO						:= 60;
//		OP90_STN_ENABLE					:= 0;
		END_IF
	
	60: IF AFT_SUP_CYL_HME.Q AND OP90_VERT_SRV_SAFE_ZONE THEN
		STATION_DONE[OP90_CURR_MOVER][OP90_XTS_POS_NO]:= TRUE;
 		OP90_STP_NO						:= 1;
		END_IF
END_CASE
END_IF


		
//////////////////////////////////HORZ/VERT SUP CYL UP//////////////////////////////////////////////
IF OP90_STN_ENABLE AND OP90_AUTO_RUNNING AND ((OP90_STP_NO=30)OR(OP90_STP_NO=35)) THEN
		IF OP90_POS1_V6_3 THEN
		OP90_A_MVR_SUP_HORZP1_HME		:= FALSE;
		OP90_A_MVR_SUP_HORZP1_WRK		:= TRUE;
		END_IF
		IF OP90_POS2_V7_89 THEN 
		OP90_A_MVR_SUP_HORZP2_HME		:= FALSE;
		OP90_A_MVR_SUP_HORZP2_WRK		:= TRUE;
		END_IF
END_IF

IF (AFT_SUP_HRZ_WRK.Q AND OP90_STP_NO<50) THEN
 	   IF OP90_POS1_V6_3 THEN
		OP90_A_MVR_SUP_VERTP1_HME		:= FALSE;
		OP90_A_MVR_SUP_VERTP1_WRK		:= TRUE;
	   END_IF
	   IF OP90_POS2_V7_89 THEN
		OP90_A_MVR_SUP_VERTP2_HME		:= FALSE;
		OP90_A_MVR_SUP_VERTP2_WRK		:= TRUE;		   
	   END_IF	
END_IF


/////////////////////////////////////////////DELAY TIMERS///////////////////////////////////////////////////////

AFT_SUP_HRZ_WRK(IN:=(OP90_POS1_V6_3 AND (I90_LH_MOVR_SUP_HORZ_CYL_FWD_I1201_1)) OR (OP90_POS2_V7_89 AND I90_RH_MOVR_SUP_HORZ_CYL_FWD_I1201_5), PT:=INT_TO_TIME(OP90_AFT_SUP_HRZ_WRK) , Q=> , ET=> );

AFT_VERT_PCK_WRK(IN:=(OP90_LH_CMP_PICKED AND NOT OP90_RH_CMP_PICKED AND OP90_SRV_RH_VRT_PCKWRK_FB) OR (NOT OP90_LH_CMP_PICKED AND  OP90_RH_CMP_PICKED AND OP90_SRV_LH_VRT_PCKWRK_FB) OR 
				(NOT OP90_LH_CMP_PICKED AND NOT OP90_RH_CMP_PICKED AND OP90_SRV_LH_VRT_PCKWRK_FB AND OP90_SRV_RH_VRT_PCKWRK_FB), PT:=INT_TO_TIME(OP90_AFT_VRT_PCK_WRK) , Q=> , ET=> );
				
AFT_PCK_DN(IN:=(OP90_STP_NO =20) AND (I90_RET_LH_GRIPR_CYL_OPN_I1200_1 OR OP90_LH_GRP_BYPASS) AND (I90_RET_RH_GRIPR_CYL_OPN_I1200_3 OR OP90_RH_GRP_BYPASS), PT:=INT_TO_TIME(OP90_AFT_CMP_PCK) , Q=> , ET=> );

AFT_VRT_PLC_WRK(IN:= (OP90_LH_CMP_OK AND NOT OP90_RH_CMP_OK AND OP90_SRV_LH_VRT_PLCWRK_FB) OR (NOT OP90_LH_CMP_OK AND  OP90_RH_CMP_OK AND OP90_SRV_RH_VRT_PLCWRK_FB)OR
					(OP90_LH_CMP_OK AND OP90_RH_CMP_OK AND OP90_SRV_LH_VRT_PLCWRK_FB AND OP90_SRV_RH_VRT_PLCWRK_FB), PT:=INT_TO_TIME(OP90_AFT_VRT_PLC_WRK) , Q=> , ET=> );
					
AFT_GRP_HME(IN:= OP90_STP_NO =50, PT:=INT_TO_TIME(OP90_AFT_GRP_HME) , Q=> , ET=> );

AFT_VRT_SUP_HME(IN:= (OP90_STP_NO =55) AND I90_LH_MOVR_SUP_VERT_CYL_DWN_I1200_6 AND I90_RH_MOVR_SUP_VERT_CYL_DWN_I1201_2  , PT:=INT_TO_TIME(OP90_AFT_SUP_VRT_HME) , Q=> , ET=> );

AFT_SUP_CYL_HME(IN:= I90_LH_MOVR_SUP_HORZ_CYL_REV_I1201_0 AND I90_RH_MOVR_SUP_HORZ_CYL_REV_I1201_4 AND OP90_SRV_LH_VRT_HME_FB AND OP90_SRV_RH_VRT_HME_FB, PT:=INT_TO_TIME(OP90_AFT_SUP_CYL_HME), Q=> , ET=> );			

ELSE
	OP90_STP_NO							:= 0;
	OP90_A_MVR_SUP_HORZP1_HME			:= FALSE;
    OP90_A_MVR_SUP_HORZP1_WRK           := FALSE;
	OP90_A_MVR_SUP_HORZP2_HME           := FALSE;
	OP90_A_MVR_SUP_HORZP2_WRK           := FALSE;
	OP90_A_MVR_SUP_VERTP1_HME		    := FALSE;
	OP90_A_MVR_SUP_VERTP1_WRK		    := FALSE;
	OP90_A_MVR_SUP_VERTP2_HME		    := FALSE;
	OP90_A_MVR_SUP_VERTP2_WRK           := FALSE;   
	OP90_A_SRV_HORZ_WRK                 := FALSE;
	OP90_A_SRV_HORZ_HME                 := FALSE;
	OP90_A_SRV_LHVERT_HME               := FALSE;
	OP90_A_SRV_LHVERT_PCKWRK            := FALSE;
	OP90_A_SRV_LHVERT_SPLCWRK           := FALSE;
	OP90_A_SRV_LHVERT_PLCWRK            := FALSE;
	OP90_A_SRV_RHVERT_HME               := FALSE;
	OP90_A_SRV_RHVERT_PCKWRK            := FALSE;
	OP90_A_SRV_RHVERT_SPLCWRK           := FALSE;
	OP90_A_SRV_RHVERT_PLCWRK            := FALSE;
	OP90_A_RH_GRP_AUTCMD2				:= FALSE;
	OP90_A_RH_GRP_AUTCMD1				:= FALSE;
	OP90_A_LH_GRP_AUTCMD2				:= FALSE;
	OP90_A_LH_GRP_AUTCMD1				:= FALSE;
	
END_IF



//####################################   	TEMP	#################################################			
				
OP90_POS1_V6_3							:= FALSE;
OP90_POS2_V7_89							:= TRUE;


//############################		OP90 STATION ENABLE CONDITION		##########################

	OP90_LH_CMP_OK						:= TRUE;
	OP90_RH_CMP_OK						:= TRUE;
	
	OP90_STN_MOVER						:= MOVER_POSITION[OP90_XTS_POS_NO];
	IF AUTO_WITH_XTS THEN	        	
	IF OP90_STN_MOVER>0 THEN   
	IF NOT(END_OF_CYCLE AND MOVER_CMP_STATUS[OP90_STN_MOVER][1]=5 AND MOVER_CMP_STATUS[OP90_STN_MOVER][2]=5)THEN	     	
	OP90_STN_ENABLE						:= MOVER_POS_RECHED[OP90_STN_MOVER] AND ((MOVER_CMP_STATUS[OP90_STN_MOVER][1]=80)OR 
											(MOVER_CMP_STATUS[OP90_STN_MOVER][2]=80)) AND STATION_ENABLE_CONTROL ;		
	ELSE
	STATION_DONE[OP90_STN_MOVER][OP90_XTS_POS_NO]			:= TRUE;		
	END_IF
	ELSE
	OP90_STN_ENABLE						:= FALSE;	
	END_IF																		
	END_IF

///////////////////////////////////// air purge ///////////////////////////
IF Track_9_TMR.Q THEN
		O90_RH_REJ_AIR_PURGE_Q1251_2 :=FALSE; 
		O90_SPARE_Q1251_3  := FALSE;
		O90_BOWL2_ENABLEQ501_1	:=0;	
ELSIF Track_10_TMR.Q OR Track_11_TMR.Q THEN
	IF Track_1_TMR.Q AND Track_5_TMR.Q AND Track_8_TMR.Q  THEN
		O90_RH_REJ_AIR_PURGE_Q1251_2 :=TRUE;
		O90_SPARE_Q1251_3  		     :=FALSE;
		O90_BOWL2_ENABLEQ501_1		 :=1;
	ELSIF Track_5_TMR.Q AND  Track_2_TMR.Q AND Track_7_TMR.Q  THEN  
		O90_SPARE_Q1251_3  			 :=TRUE;
	    O90_BOWL2_ENABLEQ501_1		 :=1;
		O90_RH_REJ_AIR_PURGE_Q1251_2 :=FALSE;
	ELSIF Track_6_TMR.Q THEN
		O90_RH_REJ_AIR_PURGE_Q1251_2 :=0; 
		O90_SPARE_Q1251_3  			 :=0;
		O90_BOWL2_ENABLEQ501_1	     :=1;		
	ELSIF Track_3_TMR.Q AND Track_9_TMR.Q THEN
		O90_RH_REJ_AIR_PURGE_Q1251_2 :=FALSE; 
		O90_SPARE_Q1251_3  			 :=FALSE;
		O90_BOWL2_ENABLEQ501_1		 :=0;	
	END_IF
END_IF

Track_1_TMR(IN:= I90_VBF1_CONV1_TRK2_OVERFLWI501_2,PT:=T#2S);
Track_2_TMR(IN:= I90_VBF1_CONV1_TRK1_OVERFLWI501_1,PT:=T#2S);
Track_3_TMR(IN:= I90_VBF1_CONV1_TRK2_OVERFLWI501_2 AND I90_VBF1_CONV1_TRK1_OVERFLWI501_1,PT:=T#2S);
Track_4_TMR(IN:= NOT I90_VBF1_CONV1_TRK2_OVERFLWI501_2 ,PT:=T#2S);
Track_5_TMR(IN:= NOT I90_VBF1_CONV1_TRK1_OVERFLWI501_1 ,PT:=T#2S);
Track_6_TMR(IN:= (NOT I90_VBF1_CONV1_TRK2_OVERFLWI501_2) AND (NOT I90_VBF1_CONV1_TRK1_OVERFLWI501_1),PT:=T#2S);

Track_7_TMR(IN:= I90_VBF1_CONV2_TRK1_OVERFLWI503_2,PT:=T#2S);
Track_8_TMR(IN:= I90_VBF1_CONV2_TRK2_OVERFLWI503_3,PT:=T#2S);
Track_9_TMR(IN:= I90_VBF1_CONV2_TRK1_OVERFLWI503_2 AND I90_VBF1_CONV2_TRK2_OVERFLWI503_3,PT:=T#2S);
Track_10_TMR(IN:= NOT I90_VBF1_CONV2_TRK1_OVERFLWI503_2 ,PT:=T#2S);
Track_11_TMR(IN:= NOT I90_VBF1_CONV2_TRK2_OVERFLWI503_3 ,PT:=T#2S);
Track_12_TMR(IN:= (NOT I90_VBF1_CONV2_TRK1_OVERFLWI503_2) AND (NOT I90_VBF1_CONV2_TRK2_OVERFLWI503_3),PT:=T#2S);

END_PROGRAM

// ---- POUs/Programs/OP90/OP90_CAMERA.TcPOU
PROGRAM OP90_CAMERA
VAR
END_VAR

OP90_LH_CMR_OK			:= TRUE;
OP90_RH_CMR_OK			:= TRUE;

END_PROGRAM

// ---- POUs/Programs/OP90/OP90_Camera_Fb.TcPOU
PROGRAM OP90_Camera_Fb
VAR
	OP90_LH_Camera 			        : FB_Cognex_ProfiNET_1;

	
	OP90_LH_Acquisition_Status AT %I*    :Acquisition_Status;
	OP90_LH_Inspection_Status  AT %I*    :Inspection_Status;	
	OP90_LH_Acquisition_ID     AT %I*    :UINT;
	OP90_LH_Inspection_ID   	 AT %I*  :UINT;
	OP90_LH_Error_code      	 AT %I*  :UINT;
	OP90_LH_Current_Job_ID  	 AT %I*  :UINT;
	OP90_LH_Result_code     	 AT %I*  :UINT;
	OP90_LH_Cam_Result      	 AT %I*  :ARRAY[0..63] OF BYTE;	
	OP90_LH_Acquisition_Control AT %Q*  : Acquisition_Control;
	OP90_LH_Inspection_Control  AT %Q*  : Inspection_Control;
	OP90_LH_Command_word		AT %Q*  : UINT;
	OP90_LH_Union                       : UNION_64Byte;

	OP90_RH_Camera 			          : FB_Cognex_ProfiNET_1;

	
	OP90_RH_Acquisition_Status AT %I*    :Acquisition_Status;
	OP90_RH_Inspection_Status  AT %I*    :Inspection_Status;	
	OP90_RH_Acquisition_ID     AT %I*    :UINT;
	OP90_RH_Inspection_ID   	 AT %I*  :UINT;
	OP90_RH_Error_code      	 AT %I*  :UINT;
	OP90_RH_Current_Job_ID  	 AT %I*  :UINT;
	OP90_RH_Result_code     	 AT %I*  :UINT;
	OP90_RH_Cam_Result      	 AT %I*  :ARRAY[0..63] OF BYTE;	
	OP90_RH_Acquisition_Control AT %Q*  : Acquisition_Control;
	OP90_RH_Inspection_Control  AT %Q*  : Inspection_Control;
	OP90_RH_Command_word		AT %Q*  : UINT;
	OP90_RH_Union                       : UNION_64Byte;	
END_VAR

OP90_LH_Camera (
	tTimeout:= , 
	sJob_Name:= , 
	camera_ready=> OP90_LH_Camera_Ready,
	Camera_online=> OP90_LH_Camera_Online,
	stCognex_record_status:=OP90_LH_Acquisition_Status, 
	Acquisition_ID:=OP90_LH_Acquisition_ID , 
	stCognex_Inspection_status:=OP90_LH_Inspection_Status, 
	Error_Code:=OP90_LH_Error_code , 
	wcommand_control_in:= OP90_LH_Current_Job_ID, 
	aResults_64_Bytes:= OP90_LH_Cam_Result, 
	number_of_inspections:=OP90_LH_Inspection_ID , 
	iresult_code:= OP90_LH_Result_code, 
	bTarget_job_ID:=OP90_LH_Target_Job_ID , 
	Error_Status_message=> OP90_LH_Error_status, 
	bError=> OP90_LH_Camera_Error, 
	stCognex_record_control=>OP90_LH_Acquisition_Control , 
	stCognex_inspection_control=>OP90_LH_Inspection_Control , 
	wCommandControl_out=>OP90_LH_Command_word , 
	aUser_data_64_Byte=> OP90_LH_Union.aArrayOfByte, 
	bJob_loading_completed=>OP90_LH_Job_Change_Complete , 
	bJob_load_failed=>OP90_LH_Job_Change_Error , 
	bInspection_Result_IO=>  , 
	bInspection_Result_NIO=> , 
	bTXTSM_Error_Job_Change=> OP90_LH_Job_Change_Error, 
	bPictureTakenComplete=> OP90_LH_Picture_Taken, 
	Loaded_Job_ID=>OP90_LH_Loaded_Job_ID	 , 
	bClear_Error:= HMI_Reset, 
	bJob_change_start:= OP90_LH_Camera_Job_Change_start, 
	TXTSM_camera_not_online=>OP90_LH_Camera_Error	 , 
	bTrigger_start:= OP90_LH_Camera_Trigger );
	
	OP90_RH_Camera (
	tTimeout:= , 
	sJob_Name:= , 
	camera_ready=> OP90_RH_Camera_Ready,
	Camera_online=> OP90_RH_Camera_Online,
	stCognex_record_status:=OP90_RH_Acquisition_Status, 
	Acquisition_ID:=OP90_RH_Acquisition_ID , 
	stCognex_Inspection_status:=OP90_RH_Inspection_Status, 
	Error_Code:=OP90_RH_Error_code , 
	wcommand_control_in:= OP90_RH_Current_Job_ID, 
	aResults_64_Bytes:= OP90_RH_Cam_Result, 
	number_of_inspections:=OP90_RH_Inspection_ID , 
	iresult_code:= OP90_RH_Result_code, 
	bTarget_job_ID:=OP90_RH_Target_Job_ID , 
	Error_Status_message=> OP90_RH_Error_status, 
	bError=> OP90_RH_Camera_Error, 
	stCognex_record_control=>OP90_RH_Acquisition_Control , 
	stCognex_inspection_control=>OP90_RH_Inspection_Control , 
	wCommandControl_out=>OP90_RH_Command_word , 
	aUser_data_64_Byte=> OP90_RH_Union.aArrayOfByte, 
	bJob_loading_completed=>OP90_RH_Job_Change_Complete , 
	bJob_load_failed=>OP90_RH_Job_Change_Error , 
	bInspection_Result_IO=>  , 
	bInspection_Result_NIO=> , 
	bTXTSM_Error_Job_Change=> OP90_RH_Job_Change_Error, 
	bPictureTakenComplete=> OP90_RH_Picture_Taken, 
	Loaded_Job_ID=>OP90_RH_Loaded_Job_ID	 , 
	bClear_Error:= HMI_Reset, 
	bJob_change_start:= OP90_RH_Camera_Job_Change_start, 
	TXTSM_camera_not_online=>OP90_RH_Camera_Error	 , 
	bTrigger_start:= OP90_RH_Camera_Trigger );

END_PROGRAM

// ---- POUs/Programs/OP90/OP90_HOMING.TcPOU
PROGRAM OP90_HOMING
VAR
// R_TRIG
	INI_R_TRIG				: R_TRIG;

// INT
	OP90_SERVO_HME_PB: BOOL;
END_VAR

IF NOT OP90_AUTO_RUNNING AND NOT OP90_STEP_RUNNING AND NOT OP90_ERR THEN 
INI_R_TRIG(CLK:= OP90_HOMING_STRT, Q=> );

IF INI_R_TRIG.Q THEN
	OP90_START_HOMNG					:= TRUE;
	OP90_HME_STP_NO						:= 1;
END_IF
	
IF OP90_START_HOMNG THEN
	CASE OP90_HME_STP_NO OF 
		1: IF OP90_LH_CMP_PICKED AND OP90_RH_CMP_PICKED THEN
			OP90_HME_STP_NO				:= 5;
			ELSIF OP90_RH_CMP_PICKED AND NOT OP90_LH_CMP_PICKED THEN
			OP90_LH_GRP_HOMING1 		:= TRUE;
			ELSIF NOT OP90_RH_CMP_PICKED AND OP90_LH_CMP_PICKED THEN
			OP90_RH_GRP_HOMING1 		:= TRUE;		
			END_IF
			OP90_HME_STP_NO				:= 5;
			
		5: IF  (OP90_LH_CMP_PICKED AND OP90_RH_CMP_PICKED)
			OR (OP90_RH_CMP_PICKED OR OP90_LH_GRIPPER.Sensor1) 
			OR (OP90_LH_CMP_PICKED OR OP90_RH_GRIPPER.Sensor1) THEN
				OP90_LH_GRP_HOMING1		:= TRUE;
				OP90_RH_GRP_HOMING1		:= TRUE;
				OP90_SERVO_HME_PB		:= TRUE;			
				OP90_HME_STP_NO			:= 15;			
			END_IF
		
		10: (*IF OP90_SRV_LH_VRT_HME_FB AND OP90_SRV_RH_VRT_HME_FB THEN
			  OP90_A_SRV_HORZ_HME			:= TRUE;
			  OP90_HME_STP_NO				:= 15;				
			END_IF*)
		
		15: IF OP90_SRV_HORZ_HME_FB THEN
			OP90_SUP_VERTP1_CYL_HOME1	:= TRUE;
			OP90_SUP_VERTP2_CYL_HOME1	:= TRUE;
			OP90_HME_STP_NO				:= 20;			
			END_IF
			
		20: IF OP90_SUP_VERTP1_CYL.Sensor1 AND OP90_SUP_VERTP2_CYL.Sensor1 THEN
			OP90_SUP_HORZP1_CYL_HOME1	:= TRUE;
			OP90_SUP_HORZP2_CYL_HOME1	:= TRUE;
			OP90_HME_STP_NO				:= 25;
			END_IF
			
		25: IF OP90_ALL_HOME THEN
			OP90_START_HOMNG					:= FALSE;
			END_IF
	END_CASE 
ELSE
	OP90_HME_STP_NO						:= 0;
	OP90_START_HOMNG							:= FALSE;
	OP90_LH_GRP_HOMING1					:= FALSE;
	OP90_RH_GRP_HOMING1					:= FALSE;
	OP90_VERT_LHSERV_HOMG1          	:= FALSE;
	OP90_HORZ_SERV_HOMING1          	:= FALSE;
	OP90_SUP_VERTP1_CYL_HOME1       	:= FALSE;
	OP90_SUP_VERTP2_CYL_HOME1	        := 0;
	OP90_SUP_HORZP1_CYL_HOME1			:= 0;
	OP90_SUP_HORZP2_CYL_HOME1			:= 0;	
	OP90_SERVO_HME_PB           		:= 0;
END_IF
END_IF

IF OP90_SERVO_HME_PB THEN
	OP90_A_SRV_HORZ_HME			:= (OP90_SRV_LH_VRT_HME_FB OR OP90_SRV_LH_VRT_ZERO_FB) AND 
									(OP90_SRV_RH_VRT_HME_FB OR OP90_SRV_RH_VRT_ZERO_FB);
	OP90_A_SRV_LH_ROTRY_HME		:= (OP90_SRV_LH_VRT_HME_FB OR OP90_SRV_LH_VRT_ZERO_FB) AND 
									(OP90_SRV_RH_VRT_HME_FB OR OP90_SRV_RH_VRT_ZERO_FB);
	OP90_A_SRV_RH_ROTRY_HME		:= (OP90_SRV_LH_VRT_HME_FB OR OP90_SRV_LH_VRT_ZERO_FB) AND 
									(OP90_SRV_RH_VRT_HME_FB OR OP90_SRV_RH_VRT_ZERO_FB);
	OP90_A_SRV_LHVERT_HME		:= TRUE;
	OP90_A_SRV_RHVERT_HME		:= TRUE;								
END_IF

//#########################  ALL HOME  #############################

IF (OP90_LH_GRIPPER.Sensor1 OR OP90_LH_CMP_PICKED) AND (OP90_RH_GRIPPER.Sensor1 OR OP90_RH_CMP_PICKED) AND
	OP90_SRV_LH_VRT_HME_FB AND OP90_SRV_RH_VRT_HME_FB AND OP90_SRV_HORZ_HME_FB AND (OP90_POS1_V6_3 OR OP90_POS2_V7_89) AND
	OP90_SUP_VERTP1_CYL.Sensor1 AND OP90_SUP_VERTP2_CYL.Sensor1 AND OP90_SUP_HORZP1_CYL.Sensor1 AND OP90_SUP_HORZP2_CYL.Sensor1 THEN
		OP90_ALL_HOME		:= TRUE;	
ELSE
		OP90_ALL_HOME		:= FALSE;
END_IF

END_PROGRAM

// ---- POUs/Programs/OP90/OP90_Conveyor_FBs.TcPOU
PROGRAM OP90_Conveyor_FBs
VAR
	OP90_Conveyor_LH 							: Servo_Conveyor_FB_OP90;
	OP90_Conveyor_RH 							: Servo_Conveyor_FB_OP90;
	
	OVR_FLW_TMR_7_89							: TON;
	OVR_FLW_TMR_6_38							: TON;
	Conveyor_Conti_run							: BOOL;
	Conveyor_Velocity_mode						: BOOL;
	OP90_Camera_Done 							: BOOL;
	OP90_One_Cycle								: BOOL;
	OP90_Conveyor_ON							: BOOL;
	OP90_RH_Conveyor_ON							: BOOL;
	OP90_LH_Conveyor_ON							: BOOL;


	BOWL_ON_OFF_7_89: TON;
	
	Conv_Cam_Step : INT :=10;
	Temp_Counter_LH : UINT;
	Temp_Counter_RH : UINT;
	Toggle_Pos: R_TRIG;
	Toggle_Neg: F_TRIG;
	Conv_Step_no: INT;
	Camera_Trigger_Ack_OP90 : BOOL;
	Toggle_Pos_LH : R_TRIG;
	Toggle_Neg_LH : F_TRIG;
	Toggle_Pos_RH : R_TRIG;
	Toggle_Neg_RH : F_TRIG;
	Track_ON_Timer: TON;
	LH_Cam_Completed : BOOL;
	RH_Cam_Completed : BOOL;	
END_VAR

VAR PERSISTENT
	OVR_FLW_TMR_7_89_TMR						: TIME;
	OVR_FLW_TMR_6_38_TMR						: TIME;	
	OP90_Conv_Fwd_Pos_7_89						: REAL;
	OP90_Conv_Rev_Pos_7_89						: REAL;
	OP90_Conveyor_FWD_Speed_7_89 				: REAL; 
	OP90_Conveyor_REV_Speed_7_89 				: REAL;
	OP90_Conv_Fwd_Pos_6_38						: REAL;
	OP90_Conv_Rev_Pos_6_38						: REAL;
	OP90_Conveyor_FWD_Speed_6_38 				: REAL; 
	OP90_Conveyor_REV_Speed_6_38 				: REAL;	
	OP90_Conv_Fwd_Time_7_89 					: INT;
	OP90_Conv_Rev_Time_7_89 					: INT;
	OP90_Conv_Fwd_Time_6_38 					: INT;
	OP90_Conv_Rev_Time_6_38 					: INT;	
	OP90_Conveyor_Manual_Speed					: REAL;	
	Track_On_Delay								: INT :=1000;
	Comp_Not_present_Counter					: INT;
	Track_Fill_Cmnd								: BOOL;
	Temp_var : BOOL;
END_VAR

Toggle_Pos_LH(CLK:=OP90_Camera_FB.OP90_LH_Inspection_Status.Inspection_Completed);
Toggle_Neg_LH(CLK:=OP90_Camera_FB.OP90_LH_Inspection_Status.Inspection_Completed);
Toggle_Pos_RH(CLK:=OP90_Camera_FB.OP90_RH_Inspection_Status.Inspection_Completed);
Toggle_Neg_RH(CLK:=OP90_Camera_FB.OP90_RH_Inspection_Status.Inspection_Completed);

IF Toggle_Pos_LH.Q OR Toggle_Neg_LH.Q THEN
	LH_Cam_Completed:=1;	
END_IF
IF Toggle_Pos_RH.Q OR Toggle_Neg_RH.Q THEN
	RH_Cam_Completed:=1;	
END_IF


IF OP90_MANUAL_SELECTED THEN               
	IF  I90_CONV1_REVI500_7 THEN
		OP90_SRV_RH_CNVY_STATUS.targetVelocity:=OP90_Conveyor_Manual_Speed;
		OP90_SRV_RH_CNVY_STATUS.moveVelocity:=TRUE;	
 	ELSIF   I90_CONV1_FWDI501_0 THEN
		OP90_SRV_RH_CNVY_STATUS.targetVelocity:=OP90_Conveyor_Manual_Speed;
		OP90_SRV_RH_CNVY_STATUS.moveVelocity:=TRUE;		
	ELSE 	
		OP90_SRV_RH_CNVY_STATUS.moveVelocity:=0;			
	END_IF  	
END_IF

IF OP90_MANUAL_SELECTED THEN               
	IF I90_CONV2_REVI503_0 THEN
		OP90_SRV_LH_CNVY_STATUS.targetVelocity:=OP90_Conveyor_Manual_Speed;
		OP90_SRV_LH_CNVY_STATUS.moveVelocity:=TRUE;
 	ELSIF I90_CONV2_FWDI503_1 THEN
		OP90_SRV_LH_CNVY_STATUS.targetVelocity:=OP90_Conveyor_Manual_Speed;
		OP90_SRV_LH_CNVY_STATUS.moveVelocity:=TRUE;		
	ELSE 	
	OP90_SRV_LH_CNVY_STATUS.moveVelocity:=0;    	
	END_IF  	
END_IF


IF (OP90_MANUAL_SELECTED AND I90_BOWL2_OFF_ONI502_6) OR (OP90_AUTO_SELECTED AND BOWL_ON_OFF_7_89.Q AND OP90_POS2_V7_89) AND NOT OP90_ERR THEN
	//O90_BOWL2_ENABLEQ501_1			:=1;
	O90_HPR2_TWR_LMP_GREENQ501_3 	:=1;
	O90_BOWL2_AIR_PURGE1Q501_4		:=1;
	O90_BOWL2_AIR_PURGE2Q501_5		:=1;
ELSE 
	O90_HPR2_TWR_LMP_GREENQ501_3 	:=0;
	//O90_BOWL2_ENABLEQ501_1			:=0;
	O90_BOWL2_AIR_PURGE1Q501_4		:=0;
	O90_BOWL2_AIR_PURGE2Q501_5		:=0;	
END_IF	

BOWL_ON_OFF_7_89(IN:= NOT (I90_VBF1_CONV2_TRK2_OVERFLWI503_3 AND I90_VBF1_CONV2_TRK1_OVERFLWI503_2), PT:=T#1S, Q=> , ET=> );


IF I90_HPR2_OFF_ONI502_7 AND NOT OP90_ERR THEN
	O90_HPR2_ENABLEQ501_0			:=1;
ELSE 
	O90_HPR2_ENABLEQ501_0			:=0;
END_IF

IF (OP90_MANUAL_SELECTED AND I90_BOWL1_OFF_ONI500_5) OR (OP90_AUTO_SELECTED AND NOT OVR_FLW_TMR_6_38.Q AND OP90_POS1_V6_3) AND NOT OP90_ERR THEN
	O90_BOWL1_ENABLEQ500_1			:=1;
	O90_HPR1_TWR_LMP_GREENQ500_3 	:=1;
	O90_BOWL1_AIR_PURGE1Q500_4		:=1;
	O90_BOWL1_AIR_PURGE2Q500_5		:=1;
ELSE 
	O90_HPR1_TWR_LMP_GREENQ500_3 	:=0;
	O90_BOWL1_ENABLEQ500_1			:=0;
	O90_BOWL1_AIR_PURGE1Q500_4		:=0;
	O90_BOWL1_AIR_PURGE2Q500_5		:=0;	
END_IF	

IF I90_HPR1_OFF_ONI500_6 AND NOT OP90_ERR THEN
	O90_HPR1_ENABLEQ500_0			:=1;
ELSE 
	O90_HPR1_ENABLEQ500_0			:=0;
END_IF


OP90_Conveyor_LH(
	Conveyor_Prgrm_Start:= OP90_LH_Conveyor_ON OR (OP90_AUTO_SELECTED AND OP90_POS2_V7_89), 
	Conveyor_Prgrm_Reset:= , 
	Conveyor_Continuous_Run:= Conveyor_Conti_run,
	Conveyor_FWD_Position	:= OP90_Conv_Fwd_Pos_7_89,
    Conveyor_REV_Position	:= OP90_Conv_Rev_Pos_7_89,
    Velocity_mode			:= Conveyor_Velocity_mode,
	Camera_Trigger_OK 	:= OP90_Camera_Done,
	Fwd_Time_IP			:= OP90_Conv_Fwd_Time_7_89, 
	Rev_Time_IP			:= OP90_Conv_Rev_Time_7_89, 
	Conveyor_FWD_Speed  := OP90_Conveyor_FWD_Speed_7_89 , 
	Conveyor_REV_Speed  := OP90_Conveyor_REV_Speed_7_89 , 
	LH_Work_Sensor:= OP90_LH_REJP2_CYL.Sensor2, 
	LH_Home_Sensor:= OP90_LH_REJP2_CYL.Sensor1, 
	RH_Work_Sensor:= OP90_RH_REJP2_CYL.Sensor2, 
	RH_Home_Sensor:=OP90_RH_REJP2_CYL.Sensor1,
	Track_Sensor_FB := Track_ON_Timer.Q, 
	Track_Overflow := OVR_FLW_TMR_7_89.Q, 
	LH_Camera_OK  := OP90_LH_Camera_OK, 
	LH_Camera_NOK := OP90_LH_Camera_NOK,
	RH_Camera_OK  := OP90_RH_Camera_OK, 
	RH_Camera_NOK := OP90_RH_Camera_NOK,
	Camera_trigger:=  OP90_CAMERA_TRIGGER, 
	LH_Work_Coil=> OP90_A_LH_REJP2_WORK, 
	LH_Home_Coil=> OP90_A_LH_REJP2_HOME, 
	RH_Work_Coil=> OP90_A_RH_REJP2_WORK,
	RH_Home_Coil=> OP90_A_RH_REJP2_HOME,
	Step_Num=> Conv_Step_no,
	Camera_Trigger_ACK=>Camera_Trigger_Ack_OP90 ,
	Ready_to_Pick=>  , 
	Pick_Done       := OP90_pick_done_7_89, 
	One_Cycle		:=  OP90_One_Cycle,
	Conveyor_Servo_Control_Structure:= OP90_SRV_LH_CNVY_CNTRL );

IF OP90_POS2_V7_89 THEN
		OP90_pick_ready					:= OP90_Conveyor_LH.Ready_to_Pick;
END_IF

OVR_FLW_TMR_7_89(IN:=I90_VBF1_CONV2_TRK2_OVERFLWI503_3 AND I90_VBF1_CONV2_TRK1_OVERFLWI503_2 , PT:=OVR_FLW_TMR_7_89_TMR, Q=> , ET=> );
Track_ON_Timer(IN:= I90_VBF1_CONV1_TRK2_OVERFLWI501_2 AND I90_VBF1_CONV1_TRK1_OVERFLWI501_1, PT:=INT_TO_TIME(Track_On_Delay), Q=> , ET=> );
	
	
	
OP90_Conveyor_RH(
	Conveyor_Prgrm_Start:= OP90_RH_Conveyor_ON OR (OP90_AUTO_SELECTED AND OP90_POS1_V6_3), 
	Conveyor_Prgrm_Reset:= , 
	Conveyor_Continuous_Run:= Conveyor_Conti_run,
	Conveyor_FWD_Position	:= OP90_Conv_Fwd_Pos_6_38,
    Conveyor_REV_Position	:= OP90_Conv_Rev_Pos_6_38,
    Velocity_mode			:= Conveyor_Velocity_mode,
	Camera_Trigger_OK   := OP90_Camera_Done,
	Fwd_Time_IP			:= OP90_Conv_Fwd_Time_6_38, 
	Rev_Time_IP			:= OP90_Conv_Rev_Time_6_38, 
	Conveyor_FWD_Speed  := OP90_Conveyor_FWD_Speed_6_38 , 
	Conveyor_REV_Speed  := OP90_Conveyor_REV_Speed_6_38 , 
	LH_Work_Sensor:= OP90_LH_REJP1_CYL.Sensor2 , 
	LH_Home_Sensor:= OP90_LH_REJP1_CYL.Sensor1, 
	RH_Work_Sensor:= OP90_RH_REJP1_CYL.Sensor2, 
	RH_Home_Sensor:=OP90_RH_REJP1_CYL.Sensor1,
	Track_Sensor_FB := Temp_var,
	Track_Overflow := OVR_FLW_TMR_6_38.Q,              
	LH_Camera_OK  := OP90_LH_Camera_OK,  
	LH_Camera_NOK := OP90_LH_Camera_NOK,
	RH_Camera_OK  := OP90_RH_Camera_OK,  
	RH_Camera_NOK := OP90_RH_Camera_NOK,
	Camera_Trigger_Ack=> OP90_Camera_Trigger_Ack,	
	Camera_trigger:=  OP90_CAMERA_TRIGGER, 
	LH_Work_Coil=> OP90_A_LH_REJP1_WORK, 
	LH_Home_Coil=> OP90_A_LH_REJP1_HOME, 
	RH_Work_Coil=>OP90_A_RH_REJP1_WORK,
	RH_Home_Coil=>OP90_A_RH_REJP1_HOME,
	Ready_to_Pick=>  , 
	Pick_Done       :=  OP90_pick_done_6_38 , 
	One_Cycle		:=  OP90_One_Cycle,
	Conveyor_Servo_Control_Structure:= OP90_SRV_RH_CNVY_CNTRL );	
	
IF OP90_POS1_V6_3 THEN
		OP90_pick_ready					:= OP90_Conveyor_RH.Ready_to_Pick;
END_IF	

OVR_FLW_TMR_6_38(IN:=I90_VBF1_CONV1_TRK2_OVERFLWI501_2 AND I90_VBF1_CONV1_TRK1_OVERFLWI501_1 , PT:=OVR_FLW_TMR_6_38_TMR, Q=> , ET=> );

IF Comp_Not_present_Counter>10 AND Track_ON_Timer.Q THEN
	//Track_Fill_Cmnd:=1;
	Comp_Not_present_Counter:=0;
END_IF

CASE Conv_Cam_Step OF
	10: 	OP90_LH_Camera_OK :=0;
            OP90_LH_Camera_NOK:=0;
	        OP90_RH_Camera_OK :=0;
	        OP90_RH_Camera_NOK:=0;	
			LH_Cam_Completed:=0;
			RH_Cam_Completed:=0;		
			OP90_Camera_Done	:=0;
			//OP90_LH_Clr_OK 		:=0;
		   // OP90_RH_Clr_OK 		:=0;		
			//OP90_LH_Size_OK		:=0;
		   // OP90_RH_Size_OK		:=0;	
			Conv_Cam_Step		:=11;	
	
